LIN {X 0,Y 425.438,Z 376.705,A -85,B 0,C 180,E1 18577.302,E2 18577.302} C_VEL
LIN {X 0,Y 425.151,Z 380.959,A -85,B 0,C 180,E1 18577.085,E2 18577.085} C_VEL
LIN {X 0,Y 415.891,Z 452.689,A -85,B 0,C 180,E1 18574.855,E2 18574.855} C_VEL
LIN {X 0,Y 409.352,Z 519.498,A -85,B 0,C 180,E1 18572.849,E2 18572.849} C_VEL
LIN {X 0,Y 405.386,Z 570.426,A -85,B 0,C 180,E1 18571.36,E2 18571.36} C_VEL
LIN {X 0,Y 403.425,Z 591.228,A -85,B 0,C 180,E1 18570.479,E2 18570.479} C_VEL
LIN {X 0,Y 401.306,Z 610.6,A -85,B 0,C 180,E1 18569.395,E2 18569.395} C_VEL
LIN {X 0,Y 398.96,Z 629.842,A -85,B 0,C 180,E1 18568.028,E2 18568.028} C_VEL
LIN {X 0,Y 396.521,Z 647.903,A -85,B 0,C 180,E1 18566.427,E2 18566.427} C_VEL
LIN {X 0,Y 394.184,Z 664.215,A -85,B 0,C 180,E1 18564.661,E2 18564.661} C_VEL
LIN {X 0,Y 391.906,Z 679.493,A -85,B 0,C 180,E1 18562.658,E2 18562.658} C_VEL
LIN {X 0,Y 389.92,Z 692.735,A -85,B 0,C 180,E1 18560.567,E2 18560.567} C_VEL
LIN {X 0,Y 388.182,Z 704.572,A -85,B 0,C 180,E1 18558.315,E2 18558.315} C_VEL
LIN {X 0,Y 386.73,Z 715.054,A -85,B 0,C 180,E1 18555.89,E2 18555.89} C_VEL
LIN {X 0,Y 385.62,Z 723.955,A -85,B 0,C 180,E1 18553.342,E2 18553.342} C_VEL
LIN {X 0,Y 384.866,Z 731.025,A -85,B 0,C 180,E1 18550.78,E2 18550.78} C_VEL
LIN {X 0,Y 384.39,Z 736.661,A -85,B 0,C 180,E1 18548.074,E2 18548.074} C_VEL
LIN {X 0,Y 384.156,Z 740.555,A -85,B 0,C 180,E1 18545.376,E2 18545.376} C_VEL
LIN {X 0,Y 384.055,Z 742.806,A -85,B 0,C 180,E1 18542.685,E2 18542.685} C_VEL
LIN {X 0,Y 384.034,Z 743.462,A -85,B 0,C 180,E1 18539.999,E2 18539.999} C_VEL
LIN {X 0,Y 384.039,Z 742.418,A -85,B 0,C 180,E1 18537.164,E2 18537.164} C_VEL
LIN {X 0,Y 384.119,Z 739.593,A -85,B 0,C 180,E1 18534.323,E2 18534.323} C_VEL
LIN {X 0,Y 384.335,Z 735.21,A -85,B 0,C 180,E1 18531.622,E2 18531.622} C_VEL
LIN {X 0,Y 384.782,Z 729.053,A -85,B 0,C 180,E1 18528.913,E2 18528.913} C_VEL
LIN {X 0,Y 385.56,Z 720.955,A -85,B 0,C 180,E1 18526.197,E2 18526.197} C_VEL
LIN {X 0,Y 386.687,Z 711.151,A -85,B 0,C 180,E1 18523.599,E2 18523.599} C_VEL
LIN {X 0,Y 388.11,Z 700.088,A -85,B 0,C 180,E1 18521.214,E2 18521.214} C_VEL
LIN {X 0,Y 389.844,Z 687.4,A -85,B 0,C 180,E1 18518.956,E2 18518.956} C_VEL
LIN {X 0,Y 391.826,Z 673.161,A -85,B 0,C 180,E1 18516.86,E2 18516.86} C_VEL
LIN {X 0,Y 393.943,Z 657.683,A -85,B 0,C 180,E1 18514.973,E2 18514.973} C_VEL
LIN {X 0,Y 396.1,Z 640.996,A -85,B 0,C 180,E1 18513.299,E2 18513.299} C_VEL
LIN {X 0,Y 398.237,Z 622.993,A -85,B 0,C 180,E1 18511.834,E2 18511.834} C_VEL
LIN {X 0,Y 400.237,Z 603.839,A -85,B 0,C 180,E1 18510.6,E2 18510.6} C_VEL
LIN {X 0,Y 401.921,Z 584.234,A -85,B 0,C 180,E1 18509.637,E2 18509.637} C_VEL
LIN {X 0,Y 403.261,Z 564.613,A -85,B 0,C 180,E1 18508.948,E2 18508.948} C_VEL
LIN {X 0,Y 404.762,Z 527.661,A -85,B 0,C 180,E1 18508.112,E2 18508.112} C_VEL
LIN {X 0,Y 410.951,Z 374.818,A -85,B 0,C 180,E1 18504.8,E2 18504.8} C_VEL
LIN {X 0,Y 406.023,Z 341.792,A -85,B 0,C 180,E1 18503.459,E2 18503.459} C_VEL
LIN {X 0,Y 404.74,Z 338.868,A -85,B 0,C 180,E1 18503.17,E2 18503.17} C_VEL
LIN {X 0,Y 398.098,Z 320.346,A -85,B 0,C 180,E1 18500.225,E2 18500.225} C_VEL
LIN {X 0,Y 390.871,Z 301.781,A -85,B 0,C 180,E1 18497.022,E2 18497.022} C_VEL
LIN {X 0,Y 385.651,Z 288.651,A -85,B 0,C 180,E1 18494.544,E2 18494.544} C_VEL
LIN {X 0,Y 385.626,Z 288.452,A -85,B 0,C 180,E1 18490.562,E2 18490.562} C_VEL
LIN {X 0,Y 385.621,Z 288.448,A -85,B 0,C 180,E1 18486.506,E2 18486.506} C_VEL
LIN {X 0,Y 385.621,Z 288.449,A -85,B 0,C 180,E1 18482.462,E2 18482.462} C_VEL
LIN {X 0,Y 385.618,Z 288.434,A -85,B 0,C 180,E1 18478.479,E2 18478.479} C_VEL
LIN {X 0,Y 385.609,Z 288.434,A -85,B 0,C 180,E1 18474.476,E2 18474.476} C_VEL
LIN {X 0,Y 385.596,Z 288.441,A -85,B 0,C 180,E1 18470.595,E2 18470.595} C_VEL
LIN {X 0,Y 385.63,Z 288.664,A -85,B 0,C 180,E1 18469.542,E2 18469.542} C_VEL
LIN {X 0,Y 388.127,Z 294.947,A -85,B 0,C 180,E1 18468.554,E2 18468.554} C_VEL
LIN {X 0,Y 395.619,Z 313.822,A -85,B 0,C 180,E1 18465.841,E2 18465.841} C_VEL
LIN {X 0,Y 402.27,Z 333.616,A -85,B 0,C 180,E1 18463.22,E2 18463.22} C_VEL
LIN {X 0,Y 402.753,Z 336.308,A -85,B 0,C 180,E1 18462.912,E2 18462.912} C_VEL
LIN {X 0,Y 402.207,Z 346.122,A -85,B 0,C 180,E1 18462.001,E2 18462.001} C_VEL
LIN {X 0,Y 400.979,Z 352.785,A -85,B 0,C 180,E1 18461.461,E2 18461.461} C_VEL
LIN {X 0,Y 394.437,Z 371.147,A -85,B 0,C 180,E1 18460.234,E2 18460.234} C_VEL
LIN {X 0,Y 393.42,Z 376.867,A -85,B 0,C 180,E1 18459.755,E2 18459.755} C_VEL
LIN {X 0,Y 390.87,Z 418.201,A -85,B 0,C 180,E1 18455.874,E2 18455.874} C_VEL
LIN {X 0,Y 388.343,Z 461.181,A -85,B 0,C 180,E1 18451.846,E2 18451.846} C_VEL
LIN {X 0,Y 387.324,Z 479.827,A -85,B 0,C 180,E1 18450.126,E2 18450.126} C_VEL
LIN {X 0,Y 389.149,Z 497.663,A -85,B 0,C 180,E1 18449.64,E2 18449.64} C_VEL
LIN {X 0,Y 386.608,Z 623.155,A -85,B 0,C 180,E1 18447.245,E2 18447.245} C_VEL
LIN {X 0,Y 385.965,Z 639.192,A -85,B 0,C 180,E1 18446.667,E2 18446.667} C_VEL
LIN {X 0,Y 384.984,Z 655.233,A -85,B 0,C 180,E1 18445.801,E2 18445.801} C_VEL
LIN {X 0,Y 383.849,Z 669.257,A -85,B 0,C 180,E1 18444.771,E2 18444.771} C_VEL
LIN {X 0,Y 382.459,Z 683.671,A -85,B 0,C 180,E1 18443.396,E2 18443.396} C_VEL
LIN {X 0,Y 381.091,Z 696.381,A -85,B 0,C 180,E1 18441.857,E2 18441.857} C_VEL
LIN {X 0,Y 379.695,Z 708.569,A -85,B 0,C 180,E1 18439.993,E2 18439.993} C_VEL
LIN {X 0,Y 378.562,Z 718.372,A -85,B 0,C 180,E1 18438.113,E2 18438.113} C_VEL
LIN {X 0,Y 377.555,Z 727.448,A -85,B 0,C 180,E1 18435.901,E2 18435.901} C_VEL
LIN {X 0,Y 376.862,Z 734.493,A -85,B 0,C 180,E1 18433.668,E2 18433.668} C_VEL
LIN {X 0,Y 376.406,Z 740.037,A -85,B 0,C 180,E1 18431.253,E2 18431.253} C_VEL
LIN {X 0,Y 376.179,Z 743.765,A -85,B 0,C 180,E1 18428.811,E2 18428.811} C_VEL
LIN {X 0,Y 376.095,Z 745.698,A -85,B 0,C 180,E1 18426.334,E2 18426.334} C_VEL
LIN {X 0,Y 376.098,Z 745.901,A -85,B 0,C 180,E1 18423.815,E2 18423.815} C_VEL
LIN {X 0,Y 376.188,Z 744.18,A -85,B 0,C 180,E1 18421.247,E2 18421.247} C_VEL
LIN {X 0,Y 376.427,Z 740.771,A -85,B 0,C 180,E1 18418.793,E2 18418.793} C_VEL
LIN {X 0,Y 376.894,Z 735.364,A -85,B 0,C 180,E1 18416.329,E2 18416.329} C_VEL
LIN {X 0,Y 377.598,Z 728.744,A -85,B 0,C 180,E1 18414.124,E2 18414.124} C_VEL
LIN {X 0,Y 378.619,Z 719.95,A -85,B 0,C 180,E1 18411.904,E2 18411.904} C_VEL
LIN {X 0,Y 379.783,Z 710.471,A -85,B 0,C 180,E1 18410.008,E2 18410.008} C_VEL
LIN {X 0,Y 381.141,Z 699.241,A -85,B 0,C 180,E1 18408.219,E2 18408.219} C_VEL
LIN {X 0,Y 382.607,Z 686.432,A -85,B 0,C 180,E1 18406.587,E2 18406.587} C_VEL
LIN {X 0,Y 383.966,Z 673.167,A -85,B 0,C 180,E1 18405.254,E2 18405.254} C_VEL
LIN {X 0,Y 385.314,Z 657.803,A -85,B 0,C 180,E1 18404.063,E2 18404.063} C_VEL
LIN {X 0,Y 386.332,Z 642.25,A -85,B 0,C 180,E1 18403.18,E2 18403.18} C_VEL
LIN {X 0,Y 387.065,Z 625.559,A -85,B 0,C 180,E1 18402.536,E2 18402.536} C_VEL
LIN {X 0,Y 387.736,Z 593.398,A -85,B 0,C 180,E1 18401.872,E2 18401.872} C_VEL
LIN {X 0,Y 389.648,Z 494.75,A -85,B 0,C 180,E1 18399.99,E2 18399.99} C_VEL
LIN {X 0,Y 387.952,Z 480.003,A -85,B 0,C 180,E1 18399.539,E2 18399.539} C_VEL
LIN {X 0,Y 390.482,Z 436.326,A -85,B 0,C 180,E1 18395.489,E2 18395.489} C_VEL
LIN {X 0,Y 393.042,Z 393.106,A -85,B 0,C 180,E1 18391.487,E2 18391.487} C_VEL
LIN {X 0,Y 395.389,Z 349.348,A -85,B 0,C 180,E1 18387.485,E2 18387.485} C_VEL
LIN {X 0,Y 396.024,Z 337.35,A -85,B 0,C 180,E1 18386.383,E2 18386.383} C_VEL
LIN {X 0,Y 390.695,Z 320.827,A -85,B 0,C 180,E1 18384.172,E2 18384.172} C_VEL
LIN {X 0,Y 384.015,Z 303.953,A -85,B 0,C 180,E1 18381.699,E2 18381.699} C_VEL
LIN {X 0,Y 378.89,Z 292.803,A -85,B 0,C 180,E1 18379.903,E2 18379.903} C_VEL
LIN {X 0,Y 377.731,Z 289.764,A -85,B 0,C 180,E1 18379.363,E2 18379.363} C_VEL
LIN {X 0,Y 377.654,Z 289.433,A -85,B 0,C 180,E1 18378.205,E2 18378.205} C_VEL
LIN {X 0,Y 377.653,Z 289.441,A -85,B 0,C 180,E1 18374.255,E2 18374.255} C_VEL
LIN {X 0,Y 377.653,Z 289.443,A -85,B 0,C 180,E1 18370.218,E2 18370.218} C_VEL
LIN {X 0,Y 377.652,Z 289.439,A -85,B 0,C 180,E1 18366.232,E2 18366.232} C_VEL
LIN {X 0,Y 377.652,Z 289.442,A -85,B 0,C 180,E1 18362.125,E2 18362.125} C_VEL
LIN {X 0,Y 377.653,Z 289.439,A -85,B 0,C 180,E1 18358.18,E2 18358.18} C_VEL
LIN {X 0,Y 377.655,Z 289.443,A -85,B 0,C 180,E1 18354.074,E2 18354.074} C_VEL
LIN {X 0,Y 377.655,Z 289.435,A -85,B 0,C 180,E1 18350.012,E2 18350.012} C_VEL
LIN {X 0,Y 377.658,Z 289.442,A -85,B 0,C 180,E1 18345.903,E2 18345.903} C_VEL
LIN {X 0,Y 377.661,Z 289.44,A -85,B 0,C 180,E1 18341.796,E2 18341.796} C_VEL
LIN {X 0,Y 377.66,Z 289.436,A -85,B 0,C 180,E1 18337.754,E2 18337.754} C_VEL
LIN {X 0,Y 377.662,Z 289.443,A -85,B 0,C 180,E1 18333.76,E2 18333.76} C_VEL
LIN {X 0,Y 377.663,Z 289.438,A -85,B 0,C 180,E1 18329.8,E2 18329.8} C_VEL
LIN {X 0,Y 377.664,Z 289.439,A -85,B 0,C 180,E1 18325.674,E2 18325.674} C_VEL
LIN {X 0,Y 377.666,Z 289.44,A -85,B 0,C 180,E1 18321.592,E2 18321.592} C_VEL
LIN {X 0,Y 377.716,Z 289.737,A -85,B 0,C 180,E1 18319.409,E2 18319.409} C_VEL
LIN {X 0,Y 386.088,Z 309.298,A -85,B 0,C 180,E1 18315.843,E2 18315.843} C_VEL
LIN {X 0,Y 390.517,Z 319.683,A -85,B 0,C 180,E1 18314.145,E2 18314.145} C_VEL
LIN {X 0,Y 407.06,Z 348.807,A -85,B 0,C 180,E1 18311.54,E2 18311.54} C_VEL
LIN {X 0,Y 409.737,Z 354.251,A -85,B 0,C 180,E1 18311.13,E2 18311.13} C_VEL
LIN {X 0,Y 401.571,Z 543.738,A -85,B 0,C 180,E1 18307.075,E2 18307.075} C_VEL
LIN {X 0,Y 399.995,Z 579.391,A -85,B 0,C 180,E1 18306.266,E2 18306.266} C_VEL
LIN {X 0,Y 398.438,Z 600.282,A -85,B 0,C 180,E1 18305.547,E2 18305.547} C_VEL
LIN {X 0,Y 396.573,Z 619.61,A -85,B 0,C 180,E1 18304.646,E2 18304.646} C_VEL
LIN {X 0,Y 394.235,Z 640.263,A -85,B 0,C 180,E1 18303.389,E2 18303.389} C_VEL
LIN {X 0,Y 391.688,Z 659.766,A -85,B 0,C 180,E1 18301.895,E2 18301.895} C_VEL
LIN {X 0,Y 389.061,Z 678.211,A -85,B 0,C 180,E1 18300.158,E2 18300.158} C_VEL
LIN {X 0,Y 386.426,Z 695.615,A -85,B 0,C 180,E1 18298.176,E2 18298.176} C_VEL
LIN {X 0,Y 384.038,Z 711.023,A -85,B 0,C 180,E1 18296.075,E2 18296.075} C_VEL
LIN {X 0,Y 381.869,Z 725.235,A -85,B 0,C 180,E1 18293.778,E2 18293.778} C_VEL
LIN {X 0,Y 379.977,Z 738.176,A -85,B 0,C 180,E1 18291.29,E2 18291.29} C_VEL
LIN {X 0,Y 378.451,Z 749.682,A -85,B 0,C 180,E1 18288.641,E2 18288.641} C_VEL
LIN {X 0,Y 377.326,Z 759.627,A -85,B 0,C 180,E1 18285.869,E2 18285.869} C_VEL
LIN {X 0,Y 376.568,Z 767.994,A -85,B 0,C 180,E1 18282.98,E2 18282.98} C_VEL
LIN {X 0,Y 376.163,Z 774.767,A -85,B 0,C 180,E1 18279.947,E2 18279.947} C_VEL
LIN {X 0,Y 376.018,Z 779.281,A -85,B 0,C 180,E1 18277.178,E2 18277.178} C_VEL
LIN {X 0,Y 376.01,Z 782.442,A -85,B 0,C 180,E1 18274.268,E2 18274.268} C_VEL
LIN {X 0,Y 376.025,Z 784,A -85,B 0,C 180,E1 18271.37,E2 18271.37} C_VEL
LIN {X 0,Y 376.03,Z 783.923,A -85,B 0,C 180,E1 18268.627,E2 18268.627} C_VEL
LIN {X 0,Y 376.014,Z 782.237,A -85,B 0,C 180,E1 18265.679,E2 18265.679} C_VEL
LIN {X 0,Y 376.027,Z 778.801,A -85,B 0,C 180,E1 18262.666,E2 18262.666} C_VEL
LIN {X 0,Y 376.183,Z 774.096,A -85,B 0,C 180,E1 18259.895,E2 18259.895} C_VEL
LIN {X 0,Y 376.573,Z 767.289,A -85,B 0,C 180,E1 18256.955,E2 18256.955} C_VEL
LIN {X 0,Y 377.294,Z 759.002,A -85,B 0,C 180,E1 18254.148,E2 18254.148} C_VEL
LIN {X 0,Y 378.404,Z 748.838,A -85,B 0,C 180,E1 18251.353,E2 18251.353} C_VEL
LIN {X 0,Y 380.005,Z 736.395,A -85,B 0,C 180,E1 18248.546,E2 18248.546} C_VEL
LIN {X 0,Y 381.94,Z 722.847,A -85,B 0,C 180,E1 18246.011,E2 18246.011} C_VEL
LIN {X 0,Y 384.155,Z 708.03,A -85,B 0,C 180,E1 18243.683,E2 18243.683} C_VEL
LIN {X 0,Y 386.6,Z 691.972,A -85,B 0,C 180,E1 18241.562,E2 18241.562} C_VEL
LIN {X 0,Y 389.239,Z 674.193,A -85,B 0,C 180,E1 18239.598,E2 18239.598} C_VEL
LIN {X 0,Y 391.918,Z 655.491,A -85,B 0,C 180,E1 18237.886,E2 18237.886} C_VEL
LIN {X 0,Y 394.591,Z 635.281,A -85,B 0,C 180,E1 18236.373,E2 18236.373} C_VEL
LIN {X 0,Y 397.071,Z 614.668,A -85,B 0,C 180,E1 18235.136,E2 18235.136} C_VEL
LIN {X 0,Y 399.349,Z 593.081,A -85,B 0,C 180,E1 18234.134,E2 18234.134} C_VEL
LIN {X 0,Y 401.355,Z 570.136,A -85,B 0,C 180,E1 18233.363,E2 18233.363} C_VEL
LIN {X 0,Y 406.419,Z 500.604,A -85,B 0,C 180,E1 18231.493,E2 18231.493} C_VEL
LIN {X 0,Y 412.494,Z 440.99,A -85,B 0,C 180,E1 18229.737,E2 18229.737} C_VEL
LIN {X 0,Y 420.617,Z 380.86,A -85,B 0,C 180,E1 18227.859,E2 18227.859} C_VEL
LIN {X 0,Y 423.847,Z 360.47,A -85,B 0,C 180,E1 18227.193,E2 18227.193} C_VEL
LIN {X 0,Y 422.14,Z 356.085,A -85,B 0,C 180,E1 18225.959,E2 18225.959} C_VEL
LIN {X 0,Y 420.779,Z 353.237,A -85,B 0,C 180,E1 18224.315,E2 18224.315} C_VEL
LIN {X 0,Y 420.316,Z 353.415,A -85,B 0,C 180,E1 18223.286,E2 18223.286} C_VEL
LIN {X 0,Y 420.495,Z 355.616,A -85,B 0,C 180,E1 18221.699,E2 18221.699} C_VEL
LIN {X 0,Y 421.439,Z 359.627,A -85,B 0,C 180,E1 18220.301,E2 18220.301} C_VEL
LIN {X 0,Y 422.49,Z 363.795,A -85,B 0,C 180,E1 18219.315,E2 18219.315} C_VEL
LIN {X 0,Y 421.522,Z 380.833,A -85,B 0,C 180,E1 18218.088,E2 18218.088} C_VEL
LIN {X 0,Y 411.493,Z 450.143,A -85,B 0,C 180,E1 18215.839,E2 18215.839} C_VEL
LIN {X 0,Y 404.087,Z 516.008,A -85,B 0,C 180,E1 18213.767,E2 18213.767} C_VEL
LIN {X 0,Y 399.163,Z 571.366,A -85,B 0,C 180,E1 18212.064,E2 18212.064} C_VEL
LIN {X 0,Y 397.052,Z 591.572,A -85,B 0,C 180,E1 18211.176,E2 18211.176} C_VEL
LIN {X 0,Y 394.706,Z 611.287,A -85,B 0,C 180,E1 18210.041,E2 18210.041} C_VEL
LIN {X 0,Y 392.165,Z 630.471,A -85,B 0,C 180,E1 18208.641,E2 18208.641} C_VEL
LIN {X 0,Y 389.562,Z 648.351,A -85,B 0,C 180,E1 18207.019,E2 18207.019} C_VEL
LIN {X 0,Y 387.063,Z 664.574,A -85,B 0,C 180,E1 18205.228,E2 18205.228} C_VEL
LIN {X 0,Y 384.714,Z 679.307,A -85,B 0,C 180,E1 18203.268,E2 18203.268} C_VEL
LIN {X 0,Y 382.565,Z 692.626,A -85,B 0,C 180,E1 18201.141,E2 18201.141} C_VEL
LIN {X 0,Y 380.677,Z 704.546,A -85,B 0,C 180,E1 18198.848,E2 18198.848} C_VEL
LIN {X 0,Y 379.096,Z 715.051,A -85,B 0,C 180,E1 18196.392,E2 18196.392} C_VEL
LIN {X 0,Y 377.852,Z 724.092,A -85,B 0,C 180,E1 18193.777,E2 18193.777} C_VEL
LIN {X 0,Y 376.99,Z 731.413,A -85,B 0,C 180,E1 18191.088,E2 18191.088} C_VEL
LIN {X 0,Y 376.472,Z 736.951,A -85,B 0,C 180,E1 18188.399,E2 18188.399} C_VEL
LIN {X 0,Y 376.195,Z 740.911,A -85,B 0,C 180,E1 18185.643,E2 18185.643} C_VEL
LIN {X 0,Y 376.078,Z 743.22,A -85,B 0,C 180,E1 18182.895,E2 18182.895} C_VEL
LIN {X 0,Y 376.045,Z 743.906,A -85,B 0,C 180,E1 18180.152,E2 18180.152} C_VEL
LIN {X 0,Y 376.045,Z 742.986,A -85,B 0,C 180,E1 18177.409,E2 18177.409} C_VEL
LIN {X 0,Y 376.115,Z 740.47,A -85,B 0,C 180,E1 18174.661,E2 18174.661} C_VEL
LIN {X 0,Y 376.317,Z 736.296,A -85,B 0,C 180,E1 18171.904,E2 18171.904} C_VEL
LIN {X 0,Y 376.755,Z 730.362,A -85,B 0,C 180,E1 18169.139,E2 18169.139} C_VEL
LIN {X 0,Y 377.502,Z 722.694,A -85,B 0,C 180,E1 18166.424,E2 18166.424} C_VEL
LIN {X 0,Y 378.557,Z 713.707,A -85,B 0,C 180,E1 18163.898,E2 18163.898} C_VEL
LIN {X 0,Y 379.979,Z 702.936,A -85,B 0,C 180,E1 18161.434,E2 18161.434} C_VEL
LIN {X 0,Y 381.705,Z 690.726,A -85,B 0,C 180,E1 18159.13,E2 18159.13} C_VEL
LIN {X 0,Y 383.685,Z 677.062,A -85,B 0,C 180,E1 18156.989,E2 18156.989} C_VEL
LIN {X 0,Y 385.869,Z 661.873,A -85,B 0,C 180,E1 18155.015,E2 18155.015} C_VEL
LIN {X 0,Y 388.085,Z 645.73,A -85,B 0,C 180,E1 18153.283,E2 18153.283} C_VEL
LIN {X 0,Y 390.283,Z 628.511,A -85,B 0,C 180,E1 18151.769,E2 18151.769} C_VEL
LIN {X 0,Y 392.391,Z 609.893,A -85,B 0,C 180,E1 18150.455,E2 18150.455} C_VEL
LIN {X 0,Y 394.273,Z 590.391,A -85,B 0,C 180,E1 18149.391,E2 18149.391} C_VEL
LIN {X 0,Y 395.803,Z 570.164,A -85,B 0,C 180,E1 18148.588,E2 18148.588} C_VEL
LIN {X 0,Y 396.936,Z 548.319,A -85,B 0,C 180,E1 18148.015,E2 18148.015} C_VEL
LIN {X 0,Y 404.242,Z 376.052,A -85,B 0,C 180,E1 18144.2,E2 18144.2} C_VEL
LIN {X 0,Y 399.757,Z 345.342,A -85,B 0,C 180,E1 18142.929,E2 18142.929} C_VEL
LIN {X 0,Y 396.829,Z 339.435,A -85,B 0,C 180,E1 18142.428,E2 18142.428} C_VEL
LIN {X 0,Y 389.659,Z 319.65,A -85,B 0,C 180,E1 18139.199,E2 18139.199} C_VEL
LIN {X 0,Y 382.005,Z 300.218,A -85,B 0,C 180,E1 18135.715,E2 18135.715} C_VEL
LIN {X 0,Y 377.705,Z 289.65,A -85,B 0,C 180,E1 18133.635,E2 18133.635} C_VEL
LIN {X 0,Y 377.684,Z 289.439,A -85,B 0,C 180,E1 18129.611,E2 18129.611} C_VEL
LIN {X 0,Y 377.682,Z 289.441,A -85,B 0,C 180,E1 18125.622,E2 18125.622} C_VEL
LIN {X 0,Y 377.683,Z 289.439,A -85,B 0,C 180,E1 18121.52,E2 18121.52} C_VEL
LIN {X 0,Y 377.673,Z 289.44,A -85,B 0,C 180,E1 18117.431,E2 18117.431} C_VEL
LIN {X 0,Y 377.665,Z 289.439,A -85,B 0,C 180,E1 18113.4,E2 18113.4} C_VEL
LIN {X 0,Y 377.702,Z 289.655,A -85,B 0,C 180,E1 18110.353,E2 18110.353} C_VEL
LIN {X 0,Y 385.933,Z 309.834,A -85,B 0,C 180,E1 18107.257,E2 18107.257} C_VEL
LIN {X 0,Y 392.695,Z 328.668,A -85,B 0,C 180,E1 18104.637,E2 18104.637} C_VEL
LIN {X 0,Y 395.707,Z 338.188,A -85,B 0,C 180,E1 18103.39,E2 18103.39} C_VEL
LIN {X 0,Y 393.42,Z 376.867,A -85,B 0,C 180,E1 18099.755,E2 18099.755} C_VEL
LIN {X 0,Y 392.128,Z 383.541,A -85,B 0,C 180,E1 18099.208,E2 18099.208} C_VEL
LIN {X 0,Y 385.455,Z 401.884,A -85,B 0,C 180,E1 18097.961,E2 18097.961} C_VEL
LIN {X 0,Y 384.433,Z 407.611,A -85,B 0,C 180,E1 18097.475,E2 18097.475} C_VEL
LIN {X 0,Y 381.606,Z 451.549,A -85,B 0,C 180,E1 18093.306,E2 18093.306} C_VEL
LIN {X 0,Y 379.974,Z 480.131,A -85,B 0,C 180,E1 18090.629,E2 18090.629} C_VEL
LIN {X 0,Y 381.841,Z 498.458,A -85,B 0,C 180,E1 18090.116,E2 18090.116} C_VEL
LIN {X 0,Y 379.17,Z 623.534,A -85,B 0,C 180,E1 18087.683,E2 18087.683} C_VEL
LIN {X 0,Y 378.494,Z 639.636,A -85,B 0,C 180,E1 18087.091,E2 18087.091} C_VEL
LIN {X 0,Y 377.466,Z 655.734,A -85,B 0,C 180,E1 18086.205,E2 18086.205} C_VEL
LIN {X 0,Y 376.243,Z 670.094,A -85,B 0,C 180,E1 18085.123,E2 18085.123} C_VEL
LIN {X 0,Y 374.792,Z 684.434,A -85,B 0,C 180,E1 18083.722,E2 18083.722} C_VEL
LIN {X 0,Y 373.359,Z 697.059,A -85,B 0,C 180,E1 18082.152,E2 18082.152} C_VEL
LIN {X 0,Y 371.897,Z 709.206,A -85,B 0,C 180,E1 18080.25,E2 18080.25} C_VEL
LIN {X 0,Y 370.678,Z 719.166,A -85,B 0,C 180,E1 18078.282,E2 18078.282} C_VEL
LIN {X 0,Y 369.647,Z 727.998,A -85,B 0,C 180,E1 18076.072,E2 18076.072} C_VEL
LIN {X 0,Y 368.914,Z 734.996,A -85,B 0,C 180,E1 18073.792,E2 18073.792} C_VEL
LIN {X 0,Y 368.428,Z 740.585,A -85,B 0,C 180,E1 18071.289,E2 18071.289} C_VEL
LIN {X 0,Y 368.192,Z 744.202,A -85,B 0,C 180,E1 18068.83,E2 18068.83} C_VEL
LIN {X 0,Y 368.104,Z 746.127,A -85,B 0,C 180,E1 18066.261,E2 18066.261} C_VEL
LIN {X 0,Y 368.109,Z 746.272,A -85,B 0,C 180,E1 18063.723,E2 18063.723} C_VEL
LIN {X 0,Y 368.211,Z 744.521,A -85,B 0,C 180,E1 18061.098,E2 18061.098} C_VEL
LIN {X 0,Y 368.472,Z 741.087,A -85,B 0,C 180,E1 18058.603,E2 18058.603} C_VEL
LIN {X 0,Y 368.99,Z 735.613,A -85,B 0,C 180,E1 18056.071,E2 18056.071} C_VEL
LIN {X 0,Y 369.729,Z 729.147,A -85,B 0,C 180,E1 18053.879,E2 18053.879} C_VEL
LIN {X 0,Y 370.786,Z 720.614,A -85,B 0,C 180,E1 18051.671,E2 18051.671} C_VEL
LIN {X 0,Y 372.085,Z 710.69,A -85,B 0,C 180,E1 18049.641,E2 18049.641} C_VEL
LIN {X 0,Y 373.545,Z 699.243,A -85,B 0,C 180,E1 18047.793,E2 18047.793} C_VEL
LIN {X 0,Y 375.103,Z 686.352,A -85,B 0,C 180,E1 18046.131,E2 18046.131} C_VEL
LIN {X 0,Y 376.6,Z 672.251,A -85,B 0,C 180,E1 18044.715,E2 18044.715} C_VEL
LIN {X 0,Y 377.97,Z 657.195,A -85,B 0,C 180,E1 18043.549,E2 18043.549} C_VEL
LIN {X 0,Y 379.05,Z 640.978,A -85,B 0,C 180,E1 18042.641,E2 18042.641} C_VEL
LIN {X 0,Y 379.755,Z 624.876,A -85,B 0,C 180,E1 18042.033,E2 18042.033} C_VEL
LIN {X 0,Y 381.195,Z 558.96,A -85,B 0,C 180,E1 18040.716,E2 18040.716} C_VEL
LIN {X 0,Y 382.467,Z 495.618,A -85,B 0,C 180,E1 18039.476,E2 18039.476} C_VEL
LIN {X 0,Y 380.711,Z 480.143,A -85,B 0,C 180,E1 18038.982,E2 18038.982} C_VEL
LIN {X 0,Y 383.378,Z 436.859,A -85,B 0,C 180,E1 18034.923,E2 18034.923} C_VEL
LIN {X 0,Y 385.959,Z 395.249,A -85,B 0,C 180,E1 18031.033,E2 18031.033} C_VEL
LIN {X 0,Y 388.328,Z 354.742,A -85,B 0,C 180,E1 18027.279,E2 18027.279} C_VEL
LIN {X 0,Y 389.068,Z 340.012,A -85,B 0,C 180,E1 18025.906,E2 18025.906} C_VEL
LIN {X 0,Y 383.738,Z 323.637,A -85,B 0,C 180,E1 18023.658,E2 18023.658} C_VEL
LIN {X 0,Y 377.887,Z 308.744,A -85,B 0,C 180,E1 18021.417,E2 18021.417} C_VEL
LIN {X 0,Y 371.317,Z 294.299,A -85,B 0,C 180,E1 18019.016,E2 18019.016} C_VEL
LIN {X 0,Y 369.768,Z 290.793,A -85,B 0,C 180,E1 18018.365,E2 18018.365} C_VEL
LIN {X 0,Y 369.741,Z 290.423,A -85,B 0,C 180,E1 18017.631,E2 18017.631} C_VEL
LIN {X 0,Y 369.751,Z 290.433,A -85,B 0,C 180,E1 18013.448,E2 18013.448} C_VEL
LIN {X 0,Y 369.746,Z 290.428,A -85,B 0,C 180,E1 18009.255,E2 18009.255} C_VEL
LIN {X 0,Y 369.746,Z 290.43,A -85,B 0,C 180,E1 18005.276,E2 18005.276} C_VEL
LIN {X 0,Y 369.746,Z 290.425,A -85,B 0,C 180,E1 18001.085,E2 18001.085} C_VEL
LIN {X 0,Y 369.741,Z 290.427,A -85,B 0,C 180,E1 17997.055,E2 17997.055} C_VEL
LIN {X 0,Y 369.746,Z 290.423,A -85,B 0,C 180,E1 17992.927,E2 17992.927} C_VEL
LIN {X 0,Y 369.735,Z 290.429,A -85,B 0,C 180,E1 17988.773,E2 17988.773} C_VEL
LIN {X 0,Y 369.742,Z 290.423,A -85,B 0,C 180,E1 17984.793,E2 17984.793} C_VEL
LIN {X 0,Y 369.737,Z 290.424,A -85,B 0,C 180,E1 17980.689,E2 17980.689} C_VEL
LIN {X 0,Y 369.735,Z 290.429,A -85,B 0,C 180,E1 17976.577,E2 17976.577} C_VEL
LIN {X 0,Y 369.731,Z 290.426,A -85,B 0,C 180,E1 17972.456,E2 17972.456} C_VEL
LIN {X 0,Y 369.733,Z 290.427,A -85,B 0,C 180,E1 17968.408,E2 17968.408} C_VEL
LIN {X 0,Y 369.727,Z 290.428,A -85,B 0,C 180,E1 17964.259,E2 17964.259} C_VEL
LIN {X 0,Y 369.775,Z 290.691,A -85,B 0,C 180,E1 17960.413,E2 17960.413} C_VEL
LIN {X 0,Y 372.529,Z 297.351,A -85,B 0,C 180,E1 17959.089,E2 17959.089} C_VEL
LIN {X 0,Y 380.514,Z 315.687,A -85,B 0,C 180,E1 17955.762,E2 17955.762} C_VEL
LIN {X 0,Y 382.502,Z 320.216,A -85,B 0,C 180,E1 17955.055,E2 17955.055} C_VEL
LIN {X 0,Y 398.543,Z 348.214,A -85,B 0,C 180,E1 17952.448,E2 17952.448} C_VEL
LIN {X 0,Y 403.094,Z 356.879,A -85,B 0,C 180,E1 17951.729,E2 17951.729} C_VEL
LIN {X 0,Y 394.051,Z 557.218,A -85,B 0,C 180,E1 17947.35,E2 17947.35} C_VEL
LIN {X 0,Y 392.751,Z 582.341,A -85,B 0,C 180,E1 17946.724,E2 17946.724} C_VEL
LIN {X 0,Y 390.974,Z 603.771,A -85,B 0,C 180,E1 17945.93,E2 17945.93} C_VEL
LIN {X 0,Y 388.828,Z 624.372,A -85,B 0,C 180,E1 17944.886,E2 17944.886} C_VEL
LIN {X 0,Y 386.349,Z 644.626,A -85,B 0,C 180,E1 17943.559,E2 17943.559} C_VEL
LIN {X 0,Y 383.787,Z 663.16,A -85,B 0,C 180,E1 17942.05,E2 17942.05} C_VEL
LIN {X 0,Y 381.235,Z 680.303,A -85,B 0,C 180,E1 17940.361,E2 17940.361} C_VEL
LIN {X 0,Y 378.598,Z 697.08,A -85,B 0,C 180,E1 17938.381,E2 17938.381} C_VEL
LIN {X 0,Y 376.01,Z 713.155,A -85,B 0,C 180,E1 17936.107,E2 17936.107} C_VEL
LIN {X 0,Y 373.725,Z 727.589,A -85,B 0,C 180,E1 17933.658,E2 17933.658} C_VEL
LIN {X 0,Y 371.736,Z 740.831,A -85,B 0,C 180,E1 17930.959,E2 17930.959} C_VEL
LIN {X 0,Y 370.249,Z 751.822,A -85,B 0,C 180,E1 17928.254,E2 17928.254} C_VEL
LIN {X 0,Y 369.161,Z 761.382,A -85,B 0,C 180,E1 17925.39,E2 17925.39} C_VEL
LIN {X 0,Y 368.458,Z 769.429,A -85,B 0,C 180,E1 17922.377,E2 17922.377} C_VEL
LIN {X 0,Y 368.119,Z 775.579,A -85,B 0,C 180,E1 17919.377,E2 17919.377} C_VEL
LIN {X 0,Y 368.022,Z 779.808,A -85,B 0,C 180,E1 17916.55,E2 17916.55} C_VEL
LIN {X 0,Y 368.02,Z 782.534,A -85,B 0,C 180,E1 17913.581,E2 17913.581} C_VEL
LIN {X 0,Y 368.043,Z 783.64,A -85,B 0,C 180,E1 17910.621,E2 17910.621} C_VEL
LIN {X 0,Y 368.035,Z 783.149,A -85,B 0,C 180,E1 17907.663,E2 17907.663} C_VEL
LIN {X 0,Y 368.011,Z 781.189,A -85,B 0,C 180,E1 17904.854,E2 17904.854} C_VEL
LIN {X 0,Y 368.069,Z 777.445,A -85,B 0,C 180,E1 17901.878,E2 17901.878} C_VEL
LIN {X 0,Y 368.282,Z 771.99,A -85,B 0,C 180,E1 17898.885,E2 17898.885} C_VEL
LIN {X 0,Y 368.805,Z 764.701,A -85,B 0,C 180,E1 17895.876,E2 17895.876} C_VEL
LIN {X 0,Y 369.691,Z 755.961,A -85,B 0,C 180,E1 17893.015,E2 17893.015} C_VEL
LIN {X 0,Y 371.059,Z 745.069,A -85,B 0,C 180,E1 17890.121,E2 17890.121} C_VEL
LIN {X 0,Y 372.804,Z 732.852,A -85,B 0,C 180,E1 17887.446,E2 17887.446} C_VEL
LIN {X 0,Y 374.959,Z 718.978,A -85,B 0,C 180,E1 17884.912,E2 17884.912} C_VEL
LIN {X 0,Y 377.339,Z 704.103,A -85,B 0,C 180,E1 17882.629,E2 17882.629} C_VEL
LIN {X 0,Y 379.992,Z 687.829,A -85,B 0,C 180,E1 17880.523,E2 17880.523} C_VEL
LIN {X 0,Y 382.806,Z 670.038,A -85,B 0,C 180,E1 17878.594,E2 17878.594} C_VEL
LIN {X 0,Y 385.753,Z 650.514,A -85,B 0,C 180,E1 17876.844,E2 17876.844} C_VEL
LIN {X 0,Y 388.648,Z 629.964,A -85,B 0,C 180,E1 17875.349,E2 17875.349} C_VEL
LIN {X 0,Y 391.397,Z 608.329,A -85,B 0,C 180,E1 17874.096,E2 17874.096} C_VEL
LIN {X 0,Y 393.844,Z 586.698,A -85,B 0,C 180,E1 17873.145,E2 17873.145} C_VEL
LIN {X 0,Y 395.974,Z 562.993,A -85,B 0,C 180,E1 17872.383,E2 17872.383} C_VEL
LIN {X 0,Y 400.952,Z 503.872,A -85,B 0,C 180,E1 17870.714,E2 17870.714} C_VEL
LIN {X 0,Y 407.588,Z 446.434,A -85,B 0,C 180,E1 17868.947,E2 17868.947} C_VEL
LIN {X 0,Y 416.346,Z 388.579,A -85,B 0,C 180,E1 17867.079,E2 17867.079} C_VEL
LIN {X 0,Y 420.44,Z 365.452,A -85,B 0,C 180,E1 17866.298,E2 17866.298} C_VEL
LIN {X 0,Y 419.53,Z 363.016,A -85,B 0,C 180,E1 17865.446,E2 17865.446} C_VEL
LIN {X 0,Y 418.737,Z 360.955,A -85,B 0,C 180,E1 17864.205,E2 17864.205} C_VEL
LIN {X 0,Y 418.331,Z 361.229,A -85,B 0,C 180,E1 17863.311,E2 17863.311} C_VEL
LIN {X 0,Y 418.348,Z 363.199,A -85,B 0,C 180,E1 17861.913,E2 17861.913} C_VEL
LIN {X 0,Y 419.16,Z 367.683,A -85,B 0,C 180,E1 17860.399,E2 17860.399} C_VEL
LIN {X 0,Y 419.383,Z 369.481,A -85,B 0,C 180,E1 17860.035,E2 17860.035} C_VEL
LIN {X 0,Y 418.006,Z 383.821,A -85,B 0,C 180,E1 17858.993,E2 17858.993} C_VEL
LIN {X 0,Y 406.652,Z 454.241,A -85,B 0,C 180,E1 17856.662,E2 17856.662} C_VEL
LIN {X 0,Y 398.55,Z 518.695,A -85,B 0,C 180,E1 17854.55,E2 17854.55} C_VEL
LIN {X 0,Y 393.19,Z 572.044,A -85,B 0,C 180,E1 17852.828,E2 17852.828} C_VEL
LIN {X 0,Y 390.813,Z 592.528,A -85,B 0,C 180,E1 17851.891,E2 17851.891} C_VEL
LIN {X 0,Y 388.137,Z 612.992,A -85,B 0,C 180,E1 17850.667,E2 17850.667} C_VEL
LIN {X 0,Y 385.32,Z 632.248,A -85,B 0,C 180,E1 17849.198,E2 17849.198} C_VEL
LIN {X 0,Y 382.563,Z 649.759,A -85,B 0,C 180,E1 17847.555,E2 17847.555} C_VEL
LIN {X 0,Y 379.805,Z 666.333,A -85,B 0,C 180,E1 17845.661,E2 17845.661} C_VEL
LIN {X 0,Y 377.138,Z 681.804,A -85,B 0,C 180,E1 17843.515,E2 17843.515} C_VEL
LIN {X 0,Y 374.817,Z 695.181,A -85,B 0,C 180,E1 17841.271,E2 17841.271} C_VEL
LIN {X 0,Y 372.735,Z 707.431,A -85,B 0,C 180,E1 17838.777,E2 17838.777} C_VEL
LIN {X 0,Y 371.118,Z 717.485,A -85,B 0,C 180,E1 17836.271,E2 17836.271} C_VEL
LIN {X 0,Y 369.861,Z 726.123,A -85,B 0,C 180,E1 17833.602,E2 17833.602} C_VEL
LIN {X 0,Y 368.975,Z 733.258,A -85,B 0,C 180,E1 17830.776,E2 17830.776} C_VEL
LIN {X 0,Y 368.446,Z 738.52,A -85,B 0,C 180,E1 17827.955,E2 17827.955} C_VEL
LIN {X 0,Y 368.187,Z 742.055,A -85,B 0,C 180,E1 17825.141,E2 17825.141} C_VEL
LIN {X 0,Y 368.078,Z 743.947,A -85,B 0,C 180,E1 17822.335,E2 17822.335} C_VEL
LIN {X 0,Y 368.051,Z 744.24,A -85,B 0,C 180,E1 17819.532,E2 17819.532} C_VEL
LIN {X 0,Y 368.066,Z 742.931,A -85,B 0,C 180,E1 17816.729,E2 17816.729} C_VEL
LIN {X 0,Y 368.166,Z 740.004,A -85,B 0,C 180,E1 17813.919,E2 17813.919} C_VEL
LIN {X 0,Y 368.438,Z 735.283,A -85,B 0,C 180,E1 17811.052,E2 17811.052} C_VEL
LIN {X 0,Y 368.976,Z 728.947,A -85,B 0,C 180,E1 17808.273,E2 17808.273} C_VEL
LIN {X 0,Y 369.827,Z 721.055,A -85,B 0,C 180,E1 17805.597,E2 17805.597} C_VEL
LIN {X 0,Y 371.003,Z 711.81,A -85,B 0,C 180,E1 17803.078,E2 17803.078} C_VEL
LIN {X 0,Y 372.593,Z 700.493,A -85,B 0,C 180,E1 17800.563,E2 17800.563} C_VEL
LIN {X 0,Y 374.5,Z 687.664,A -85,B 0,C 180,E1 17798.215,E2 17798.215} C_VEL
LIN {X 0,Y 376.673,Z 673.272,A -85,B 0,C 180,E1 17796.037,E2 17796.037} C_VEL
LIN {X 0,Y 378.915,Z 658.124,A -85,B 0,C 180,E1 17794.135,E2 17794.135} C_VEL
LIN {X 0,Y 381.192,Z 641.872,A -85,B 0,C 180,E1 17792.447,E2 17792.447} C_VEL
LIN {X 0,Y 383.414,Z 624.653,A -85,B 0,C 180,E1 17790.984,E2 17790.984} C_VEL
LIN {X 0,Y 385.514,Z 606.259,A -85,B 0,C 180,E1 17789.732,E2 17789.732} C_VEL
LIN {X 0,Y 387.38,Z 586.654,A -85,B 0,C 180,E1 17788.703,E2 17788.703} C_VEL
LIN {X 0,Y 388.941,Z 566.164,A -85,B 0,C 180,E1 17787.931,E2 17787.931} C_VEL
LIN {X 0,Y 390.345,Z 536.46,A -85,B 0,C 180,E1 17787.204,E2 17787.204} C_VEL
LIN {X 0,Y 397.577,Z 377.275,A -85,B 0,C 180,E1 17783.581,E2 17783.581} C_VEL
LIN {X 0,Y 393.441,Z 348.721,A -85,B 0,C 180,E1 17782.369,E2 17782.369} C_VEL
LIN {X 0,Y 388.564,Z 339.103,A -85,B 0,C 180,E1 17781.529,E2 17781.529} C_VEL
LIN {X 0,Y 381.373,Z 319.703,A -85,B 0,C 180,E1 17778.246,E2 17778.246} C_VEL
LIN {X 0,Y 374.161,Z 301.415,A -85,B 0,C 180,E1 17774.87,E2 17774.87} C_VEL
LIN {X 0,Y 369.778,Z 290.655,A -85,B 0,C 180,E1 17772.684,E2 17772.684} C_VEL
LIN {X 0,Y 369.749,Z 290.429,A -85,B 0,C 180,E1 17768.601,E2 17768.601} C_VEL
LIN {X 0,Y 369.743,Z 290.426,A -85,B 0,C 180,E1 17764.416,E2 17764.416} C_VEL
LIN {X 0,Y 369.747,Z 290.411,A -85,B 0,C 180,E1 17760.378,E2 17760.378} C_VEL
LIN {X 0,Y 369.739,Z 290.421,A -85,B 0,C 180,E1 17756.328,E2 17756.328} C_VEL
LIN {X 0,Y 369.744,Z 290.418,A -85,B 0,C 180,E1 17752.248,E2 17752.248} C_VEL
LIN {X 0,Y 369.75,Z 290.681,A -85,B 0,C 180,E1 17751.205,E2 17751.205} C_VEL
LIN {X 0,Y 378.347,Z 311.374,A -85,B 0,C 180,E1 17747.939,E2 17747.939} C_VEL
LIN {X 0,Y 385.096,Z 329.918,A -85,B 0,C 180,E1 17745.281,E2 17745.281} C_VEL
LIN {X 0,Y 388.637,Z 341.241,A -85,B 0,C 180,E1 17743.769,E2 17743.769} C_VEL
LIN {X 0,Y 386.021,Z 382.579,A -85,B 0,C 180,E1 17739.845,E2 17739.845} C_VEL
LIN {X 0,Y 384.433,Z 407.611,A -85,B 0,C 180,E1 17737.475,E2 17737.475} C_VEL
LIN {X 0,Y 383.132,Z 414.289,A -85,B 0,C 180,E1 17736.917,E2 17736.917} C_VEL
LIN {X 0,Y 376.341,Z 432.592,A -85,B 0,C 180,E1 17735.645,E2 17735.645} C_VEL
LIN {X 0,Y 375.3,Z 438.327,A -85,B 0,C 180,E1 17735.151,E2 17735.151} C_VEL
LIN {X 0,Y 372.631,Z 480.345,A -85,B 0,C 180,E1 17731.15,E2 17731.15} C_VEL
LIN {X 0,Y 374.555,Z 499.287,A -85,B 0,C 180,E1 17730.609,E2 17730.609} C_VEL
LIN {X 0,Y 371.744,Z 623.954,A -85,B 0,C 180,E1 17728.133,E2 17728.133} C_VEL
LIN {X 0,Y 371.04,Z 640.012,A -85,B 0,C 180,E1 17727.531,E2 17727.531} C_VEL
LIN {X 0,Y 369.982,Z 655.877,A -85,B 0,C 180,E1 17726.643,E2 17726.643} C_VEL
LIN {X 0,Y 368.737,Z 669.994,A -85,B 0,C 180,E1 17725.57,E2 17725.57} C_VEL
LIN {X 0,Y 367.225,Z 684.313,A -85,B 0,C 180,E1 17724.154,E2 17724.154} C_VEL
LIN {X 0,Y 365.703,Z 697.159,A -85,B 0,C 180,E1 17722.54,E2 17722.54} C_VEL
LIN {X 0,Y 364.22,Z 708.895,A -85,B 0,C 180,E1 17720.681,E2 17720.681} C_VEL
LIN {X 0,Y 362.949,Z 718.813,A -85,B 0,C 180,E1 17718.723,E2 17718.723} C_VEL
LIN {X 0,Y 361.809,Z 727.957,A -85,B 0,C 180,E1 17716.416,E2 17716.416} C_VEL
LIN {X 0,Y 361.014,Z 735.082,A -85,B 0,C 180,E1 17714.088,E2 17714.088} C_VEL
LIN {X 0,Y 360.481,Z 740.708,A -85,B 0,C 180,E1 17711.552,E2 17711.552} C_VEL
LIN {X 0,Y 360.22,Z 744.468,A -85,B 0,C 180,E1 17709.021,E2 17709.021} C_VEL
LIN {X 0,Y 360.115,Z 746.468,A -85,B 0,C 180,E1 17706.385,E2 17706.385} C_VEL
LIN {X 0,Y 360.118,Z 746.707,A -85,B 0,C 180,E1 17703.805,E2 17703.805} C_VEL
LIN {X 0,Y 360.212,Z 745.207,A -85,B 0,C 180,E1 17701.301,E2 17701.301} C_VEL
LIN {X 0,Y 360.482,Z 741.88,A -85,B 0,C 180,E1 17698.683,E2 17698.683} C_VEL
LIN {X 0,Y 360.99,Z 736.788,A -85,B 0,C 180,E1 17696.173,E2 17696.173} C_VEL
LIN {X 0,Y 361.814,Z 729.961,A -85,B 0,C 180,E1 17693.748,E2 17693.748} C_VEL
LIN {X 0,Y 362.929,Z 721.526,A -85,B 0,C 180,E1 17691.483,E2 17691.483} C_VEL
LIN {X 0,Y 364.342,Z 711.321,A -85,B 0,C 180,E1 17689.337,E2 17689.337} C_VEL
LIN {X 0,Y 365.805,Z 700.533,A -85,B 0,C 180,E1 17687.539,E2 17687.539} C_VEL
LIN {X 0,Y 367.422,Z 687.824,A -85,B 0,C 180,E1 17685.844,E2 17685.844} C_VEL
LIN {X 0,Y 368.904,Z 674.932,A -85,B 0,C 180,E1 17684.477,E2 17684.477} C_VEL
LIN {X 0,Y 370.302,Z 660.652,A -85,B 0,C 180,E1 17683.302,E2 17683.302} C_VEL
LIN {X 0,Y 371.494,Z 645.139,A -85,B 0,C 180,E1 17682.341,E2 17682.341} C_VEL
LIN {X 0,Y 372.331,Z 628.571,A -85,B 0,C 180,E1 17681.645,E2 17681.645} C_VEL
LIN {X 0,Y 372.829,Z 609.797,A -85,B 0,C 180,E1 17681.189,E2 17681.189} C_VEL
LIN {X 0,Y 375.331,Z 496.579,A -85,B 0,C 180,E1 17678.943,E2 17678.943} C_VEL
LIN {X 0,Y 373.529,Z 480.228,A -85,B 0,C 180,E1 17678.391,E2 17678.391} C_VEL
LIN {X 0,Y 376.355,Z 437.011,A -85,B 0,C 180,E1 17674.291,E2 17674.291} C_VEL
LIN {X 0,Y 379.094,Z 395.27,A -85,B 0,C 180,E1 17670.346,E2 17670.346} C_VEL
LIN {X 0,Y 381.738,Z 352.371,A -85,B 0,C 180,E1 17666.329,E2 17666.329} C_VEL
LIN {X 0,Y 382.179,Z 342.798,A -85,B 0,C 180,E1 17665.408,E2 17665.408} C_VEL
LIN {X 0,Y 376.531,Z 325.559,A -85,B 0,C 180,E1 17662.977,E2 17662.977} C_VEL
LIN {X 0,Y 370.306,Z 310.03,A -85,B 0,C 180,E1 17660.55,E2 17660.55} C_VEL
LIN {X 0,Y 364.847,Z 298.49,A -85,B 0,C 180,E1 17658.536,E2 17658.536} C_VEL
LIN {X 0,Y 361.863,Z 291.816,A -85,B 0,C 180,E1 17657.28,E2 17657.28} C_VEL
LIN {X 0,Y 361.776,Z 291.421,A -85,B 0,C 180,E1 17656.705,E2 17656.705} C_VEL
LIN {X 0,Y 361.777,Z 291.421,A -85,B 0,C 180,E1 17652.612,E2 17652.612} C_VEL
LIN {X 0,Y 361.775,Z 291.418,A -85,B 0,C 180,E1 17648.424,E2 17648.424} C_VEL
LIN {X 0,Y 361.776,Z 291.417,A -85,B 0,C 180,E1 17644.28,E2 17644.28} C_VEL
LIN {X 0,Y 361.777,Z 291.421,A -85,B 0,C 180,E1 17640.159,E2 17640.159} C_VEL
LIN {X 0,Y 361.777,Z 291.414,A -85,B 0,C 180,E1 17636.039,E2 17636.039} C_VEL
LIN {X 0,Y 361.78,Z 291.42,A -85,B 0,C 180,E1 17631.898,E2 17631.898} C_VEL
LIN {X 0,Y 361.786,Z 291.414,A -85,B 0,C 180,E1 17627.714,E2 17627.714} C_VEL
LIN {X 0,Y 361.79,Z 291.413,A -85,B 0,C 180,E1 17623.627,E2 17623.627} C_VEL
LIN {X 0,Y 361.799,Z 291.42,A -85,B 0,C 180,E1 17619.454,E2 17619.454} C_VEL
LIN {X 0,Y 361.801,Z 291.414,A -85,B 0,C 180,E1 17615.336,E2 17615.336} C_VEL
LIN {X 0,Y 361.818,Z 291.415,A -85,B 0,C 180,E1 17611.08,E2 17611.08} C_VEL
LIN {X 0,Y 361.809,Z 291.418,A -85,B 0,C 180,E1 17606.856,E2 17606.856} C_VEL
LIN {X 0,Y 361.808,Z 291.417,A -85,B 0,C 180,E1 17602.735,E2 17602.735} C_VEL
LIN {X 0,Y 361.853,Z 291.791,A -85,B 0,C 180,E1 17601.399,E2 17601.399} C_VEL
LIN {X 0,Y 370.051,Z 310.673,A -85,B 0,C 180,E1 17597.718,E2 17597.718} C_VEL
LIN {X 0,Y 374.269,Z 320.363,A -85,B 0,C 180,E1 17596.033,E2 17596.033} C_VEL
LIN {X 0,Y 391.264,Z 349.93,A -85,B 0,C 180,E1 17593.176,E2 17593.176} C_VEL
LIN {X 0,Y 396.467,Z 359.906,A -85,B 0,C 180,E1 17592.338,E2 17592.338} C_VEL
LIN {X 0,Y 387.034,Z 557.79,A -85,B 0,C 180,E1 17587.909,E2 17587.909} C_VEL
LIN {X 0,Y 385.672,Z 582.621,A -85,B 0,C 180,E1 17587.271,E2 17587.271} C_VEL
LIN {X 0,Y 383.819,Z 604.013,A -85,B 0,C 180,E1 17586.458,E2 17586.458} C_VEL
LIN {X 0,Y 381.572,Z 624.706,A -85,B 0,C 180,E1 17585.385,E2 17585.385} C_VEL
LIN {X 0,Y 378.957,Z 645.216,A -85,B 0,C 180,E1 17584.008,E2 17584.008} C_VEL
LIN {X 0,Y 376.163,Z 664.59,A -85,B 0,C 180,E1 17582.382,E2 17582.382} C_VEL
LIN {X 0,Y 373.295,Z 682.905,A -85,B 0,C 180,E1 17580.5,E2 17580.5} C_VEL
LIN {X 0,Y 370.468,Z 700.128,A -85,B 0,C 180,E1 17578.357,E2 17578.357} C_VEL
LIN {X 0,Y 367.863,Z 715.674,A -85,B 0,C 180,E1 17576.035,E2 17576.035} C_VEL
LIN {X 0,Y 365.568,Z 729.69,A -85,B 0,C 180,E1 17573.534,E2 17573.534} C_VEL
LIN {X 0,Y 363.692,Z 741.895,A -85,B 0,C 180,E1 17570.938,E2 17570.938} C_VEL
LIN {X 0,Y 362.195,Z 752.719,A -85,B 0,C 180,E1 17568.174,E2 17568.174} C_VEL
LIN {X 0,Y 361.109,Z 762.048,A -85,B 0,C 180,E1 17565.249,E2 17565.249} C_VEL
LIN {X 0,Y 360.45,Z 769.492,A -85,B 0,C 180,E1 17562.331,E2 17562.331} C_VEL
LIN {X 0,Y 360.116,Z 775.518,A -85,B 0,C 180,E1 17559.265,E2 17559.265} C_VEL
LIN {X 0,Y 360.029,Z 779.619,A -85,B 0,C 180,E1 17556.376,E2 17556.376} C_VEL
LIN {X 0,Y 360.031,Z 782.152,A -85,B 0,C 180,E1 17553.501,E2 17553.501} C_VEL
LIN {X 0,Y 360.056,Z 783.184,A -85,B 0,C 180,E1 17550.635,E2 17550.635} C_VEL
LIN {X 0,Y 360.046,Z 782.801,A -85,B 0,C 180,E1 17547.77,E2 17547.77} C_VEL
LIN {X 0,Y 360.019,Z 780.891,A -85,B 0,C 180,E1 17544.9,E2 17544.9} C_VEL
LIN {X 0,Y 360.071,Z 777.255,A -85,B 0,C 180,E1 17541.857,E2 17541.857} C_VEL
LIN {X 0,Y 360.29,Z 771.904,A -85,B 0,C 180,E1 17538.797,E2 17538.797} C_VEL
LIN {X 0,Y 360.802,Z 765.169,A -85,B 0,C 180,E1 17535.884,E2 17535.884} C_VEL
LIN {X 0,Y 361.715,Z 756.614,A -85,B 0,C 180,E1 17532.96,E2 17532.96} C_VEL
LIN {X 0,Y 363.113,Z 746.047,A -85,B 0,C 180,E1 17530.034,E2 17530.034} C_VEL
LIN {X 0,Y 364.945,Z 733.976,A -85,B 0,C 180,E1 17527.274,E2 17527.274} C_VEL
LIN {X 0,Y 367.19,Z 720.436,A -85,B 0,C 180,E1 17524.689,E2 17524.689} C_VEL
LIN {X 0,Y 369.866,Z 704.884,A -85,B 0,C 180,E1 17522.203,E2 17522.203} C_VEL
LIN {X 0,Y 372.777,Z 688.278,A -85,B 0,C 180,E1 17519.983,E2 17519.983} C_VEL
LIN {X 0,Y 375.897,Z 670.021,A -85,B 0,C 180,E1 17517.949,E2 17517.949} C_VEL
LIN {X 0,Y 379.18,Z 649.853,A -85,B 0,C 180,E1 17516.101,E2 17516.101} C_VEL
LIN {X 0,Y 382.324,Z 629.271,A -85,B 0,C 180,E1 17514.573,E2 17514.573} C_VEL
LIN {X 0,Y 385.372,Z 607.362,A -85,B 0,C 180,E1 17513.278,E2 17513.278} C_VEL
LIN {X 0,Y 388.095,Z 585.513,A -85,B 0,C 180,E1 17512.297,E2 17512.297} C_VEL
LIN {X 0,Y 390.531,Z 561.018,A -85,B 0,C 180,E1 17511.491,E2 17511.491} C_VEL
LIN {X 0,Y 396.15,Z 504.027,A -85,B 0,C 180,E1 17509.79,E2 17509.79} C_VEL
LIN {X 0,Y 403.596,Z 448.199,A -85,B 0,C 180,E1 17507.993,E2 17507.993} C_VEL
LIN {X 0,Y 413.32,Z 391.687,A -85,B 0,C 180,E1 17506.113,E2 17506.113} C_VEL
LIN {X 0,Y 417.462,Z 370.843,A -85,B 0,C 180,E1 17505.397,E2 17505.397} C_VEL
LIN {X 0,Y 416.625,Z 368.637,A -85,B 0,C 180,E1 17503.947,E2 17503.947} C_VEL
LIN {X 0,Y 416.23,Z 370.282,A -85,B 0,C 180,E1 17502.352,E2 17502.352} C_VEL
LIN {X 0,Y 416.609,Z 374.396,A -85,B 0,C 180,E1 17500.886,E2 17500.886} C_VEL
LIN {X 0,Y 416.295,Z 377.115,A -85,B 0,C 180,E1 17500.625,E2 17500.625} C_VEL
LIN {X 0,Y 414.994,Z 386.565,A -85,B 0,C 180,E1 17499.964,E2 17499.964} C_VEL
LIN {X 0,Y 402.614,Z 455.585,A -85,B 0,C 180,E1 17497.622,E2 17497.622} C_VEL
LIN {X 0,Y 393.658,Z 518.567,A -85,B 0,C 180,E1 17495.476,E2 17495.476} C_VEL
LIN {X 0,Y 387.47,Z 572.808,A -85,B 0,C 180,E1 17493.641,E2 17493.641} C_VEL
LIN {X 0,Y 384.736,Z 593.941,A -85,B 0,C 180,E1 17492.632,E2 17492.632} C_VEL
LIN {X 0,Y 381.83,Z 613.98,A -85,B 0,C 180,E1 17491.386,E2 17491.386} C_VEL
LIN {X 0,Y 378.704,Z 633.508,A -85,B 0,C 180,E1 17489.846,E2 17489.846} C_VEL
LIN {X 0,Y 375.638,Z 651.411,A -85,B 0,C 180,E1 17488.107,E2 17488.107} C_VEL
LIN {X 0,Y 372.601,Z 668.27,A -85,B 0,C 180,E1 17486.109,E2 17486.109} C_VEL
LIN {X 0,Y 369.779,Z 683.433,A -85,B 0,C 180,E1 17483.928,E2 17483.928} C_VEL
LIN {X 0,Y 367.393,Z 696.148,A -85,B 0,C 180,E1 17481.723,E2 17481.723} C_VEL
LIN {X 0,Y 365.287,Z 707.58,A -85,B 0,C 180,E1 17479.341,E2 17479.341} C_VEL
LIN {X 0,Y 363.518,Z 717.679,A -85,B 0,C 180,E1 17476.786,E2 17476.786} C_VEL
LIN {X 0,Y 362.121,Z 726.367,A -85,B 0,C 180,E1 17474.062,E2 17474.062} C_VEL
LIN {X 0,Y 361.126,Z 733.552,A -85,B 0,C 180,E1 17471.175,E2 17471.175} C_VEL
LIN {X 0,Y 360.532,Z 738.865,A -85,B 0,C 180,E1 17468.291,E2 17468.291} C_VEL
LIN {X 0,Y 360.229,Z 742.445,A -85,B 0,C 180,E1 17465.415,E2 17465.415} C_VEL
LIN {X 0,Y 360.095,Z 744.439,A -85,B 0,C 180,E1 17462.386,E2 17462.386} C_VEL
LIN {X 0,Y 360.063,Z 744.673,A -85,B 0,C 180,E1 17459.522,E2 17459.522} C_VEL
LIN {X 0,Y 360.078,Z 743.299,A -85,B 0,C 180,E1 17456.656,E2 17456.656} C_VEL
LIN {X 0,Y 360.185,Z 740.297,A -85,B 0,C 180,E1 17453.784,E2 17453.784} C_VEL
LIN {X 0,Y 360.473,Z 735.589,A -85,B 0,C 180,E1 17450.903,E2 17450.903} C_VEL
LIN {X 0,Y 361.018,Z 729.481,A -85,B 0,C 180,E1 17448.173,E2 17448.173} C_VEL
LIN {X 0,Y 361.907,Z 721.59,A -85,B 0,C 180,E1 17445.438,E2 17445.438} C_VEL
LIN {X 0,Y 363.22,Z 711.678,A -85,B 0,C 180,E1 17442.704,E2 17442.704} C_VEL
LIN {X 0,Y 364.906,Z 700.221,A -85,B 0,C 180,E1 17440.137,E2 17440.137} C_VEL
LIN {X 0,Y 366.92,Z 687.23,A -85,B 0,C 180,E1 17437.741,E2 17437.741} C_VEL
LIN {X 0,Y 369.206,Z 672.655,A -85,B 0,C 180,E1 17435.521,E2 17435.521} C_VEL
LIN {X 0,Y 371.695,Z 656.362,A -85,B 0,C 180,E1 17433.477,E2 17433.477} C_VEL
LIN {X 0,Y 374.101,Z 639.723,A -85,B 0,C 180,E1 17431.766,E2 17431.766} C_VEL
LIN {X 0,Y 376.392,Z 622.31,A -85,B 0,C 180,E1 17430.304,E2 17430.304} C_VEL
LIN {X 0,Y 378.516,Z 604.11,A -85,B 0,C 180,E1 17429.084,E2 17429.084} C_VEL
LIN {X 0,Y 380.423,Z 584.401,A -85,B 0,C 180,E1 17428.065,E2 17428.065} C_VEL
LIN {X 0,Y 381.947,Z 564.641,A -85,B 0,C 180,E1 17427.332,E2 17427.332} C_VEL
LIN {X 0,Y 384.109,Z 518.749,A -85,B 0,C 180,E1 17426.225,E2 17426.225} C_VEL
LIN {X 0,Y 390.905,Z 378.386,A -85,B 0,C 180,E1 17422.945,E2 17422.945} C_VEL
LIN {X 0,Y 387.233,Z 352.342,A -85,B 0,C 180,E1 17421.807,E2 17421.807} C_VEL
LIN {X 0,Y 380.321,Z 338.936,A -85,B 0,C 180,E1 17420.619,E2 17420.619} C_VEL
LIN {X 0,Y 372.972,Z 319.156,A -85,B 0,C 180,E1 17417.157,E2 17417.157} C_VEL
LIN {X 0,Y 365.795,Z 301.475,A -85,B 0,C 180,E1 17413.754,E2 17413.754} C_VEL
LIN {X 0,Y 361.828,Z 291.608,A -85,B 0,C 180,E1 17411.679,E2 17411.679} C_VEL
LIN {X 0,Y 361.805,Z 291.418,A -85,B 0,C 180,E1 17407.52,E2 17407.52} C_VEL
LIN {X 0,Y 361.803,Z 291.417,A -85,B 0,C 180,E1 17403.365,E2 17403.365} C_VEL
LIN {X 0,Y 361.793,Z 291.394,A -85,B 0,C 180,E1 17399.287,E2 17399.287} C_VEL
LIN {X 0,Y 361.781,Z 291.399,A -85,B 0,C 180,E1 17395.191,E2 17395.191} C_VEL
LIN {X 0,Y 361.849,Z 291.658,A -85,B 0,C 180,E1 17392.118,E2 17392.118} C_VEL
LIN {X 0,Y 364.914,Z 298.892,A -85,B 0,C 180,E1 17390.877,E2 17390.877} C_VEL
LIN {X 0,Y 372.715,Z 317.86,A -85,B 0,C 180,E1 17387.89,E2 17387.89} C_VEL
LIN {X 0,Y 379.259,Z 336.41,A -85,B 0,C 180,E1 17385.222,E2 17385.222} C_VEL
LIN {X 0,Y 381.599,Z 344.037,A -85,B 0,C 180,E1 17384.192,E2 17384.192} C_VEL
LIN {X 0,Y 378.865,Z 384.794,A -85,B 0,C 180,E1 17380.278,E2 17380.278} C_VEL
LIN {X 0,Y 376.074,Z 426.012,A -85,B 0,C 180,E1 17376.336,E2 17376.336} C_VEL
LIN {X 0,Y 375.3,Z 438.327,A -85,B 0,C 180,E1 17375.151,E2 17375.151} C_VEL
LIN {X 0,Y 373.99,Z 445.018,A -85,B 0,C 180,E1 17374.584,E2 17374.584} C_VEL
LIN {X 0,Y 367.132,Z 463.306,A -85,B 0,C 180,E1 17373.284,E2 17373.284} C_VEL
LIN {X 0,Y 366.041,Z 469.044,A -85,B 0,C 180,E1 17372.779,E2 17372.779} C_VEL
LIN {X 0,Y 365.34,Z 480.845,A -85,B 0,C 180,E1 17371.678,E2 17371.678} C_VEL
LIN {X 0,Y 367.274,Z 500.091,A -85,B 0,C 180,E1 17371.113,E2 17371.113} C_VEL
LIN {X 0,Y 364.343,Z 624.371,A -85,B 0,C 180,E1 17368.601,E2 17368.601} C_VEL
LIN {X 0,Y 363.607,Z 640.39,A -85,B 0,C 180,E1 17367.989,E2 17367.989} C_VEL
LIN {X 0,Y 362.484,Z 656.498,A -85,B 0,C 180,E1 17367.069,E2 17367.069} C_VEL
LIN {X 0,Y 361.159,Z 670.777,A -85,B 0,C 180,E1 17365.954,E2 17365.954} C_VEL
LIN {X 0,Y 359.596,Z 684.917,A -85,B 0,C 180,E1 17364.523,E2 17364.523} C_VEL
LIN {X 0,Y 358.065,Z 697.249,A -85,B 0,C 180,E1 17362.944,E2 17362.944} C_VEL
LIN {X 0,Y 356.414,Z 709.709,A -85,B 0,C 180,E1 17360.927,E2 17360.927} C_VEL
LIN {X 0,Y 355.108,Z 719.37,A -85,B 0,C 180,E1 17358.964,E2 17358.964} C_VEL
LIN {X 0,Y 353.909,Z 728.488,A -85,B 0,C 180,E1 17356.607,E2 17356.607} C_VEL
LIN {X 0,Y 353.071,Z 735.573,A -85,B 0,C 180,E1 17354.227,E2 17354.227} C_VEL
LIN {X 0,Y 352.513,Z 741.144,A -85,B 0,C 180,E1 17351.651,E2 17351.651} C_VEL
LIN {X 0,Y 352.233,Z 744.901,A -85,B 0,C 180,E1 17349.045,E2 17349.045} C_VEL
LIN {X 0,Y 352.125,Z 746.856,A -85,B 0,C 180,E1 17346.401,E2 17346.401} C_VEL
LIN {X 0,Y 352.13,Z 747.086,A -85,B 0,C 180,E1 17343.71,E2 17343.71} C_VEL
LIN {X 0,Y 352.235,Z 745.556,A -85,B 0,C 180,E1 17341.149,E2 17341.149} C_VEL
LIN {X 0,Y 352.521,Z 742.31,A -85,B 0,C 180,E1 17338.544,E2 17338.544} C_VEL
LIN {X 0,Y 353.041,Z 737.486,A -85,B 0,C 180,E1 17336.081,E2 17336.081} C_VEL
LIN {X 0,Y 353.901,Z 730.768,A -85,B 0,C 180,E1 17333.611,E2 17333.611} C_VEL
LIN {X 0,Y 355.064,Z 722.531,A -85,B 0,C 180,E1 17331.31,E2 17331.31} C_VEL
LIN {X 0,Y 356.577,Z 712.182,A -85,B 0,C 180,E1 17329.063,E2 17329.063} C_VEL
LIN {X 0,Y 358.152,Z 701.269,A -85,B 0,C 180,E1 17327.187,E2 17327.187} C_VEL
LIN {X 0,Y 359.962,Z 687.793,A -85,B 0,C 180,E1 17325.355,E2 17325.355} C_VEL
LIN {X 0,Y 361.603,Z 674.011,A -85,B 0,C 180,E1 17323.893,E2 17323.893} C_VEL
LIN {X 0,Y 363.109,Z 659.138,A -85,B 0,C 180,E1 17322.678,E2 17322.678} C_VEL
LIN {X 0,Y 364.287,Z 643.643,A -85,B 0,C 180,E1 17321.746,E2 17321.746} C_VEL
LIN {X 0,Y 365.139,Z 626.953,A -85,B 0,C 180,E1 17321.063,E2 17321.063} C_VEL
LIN {X 0,Y 365.879,Z 597.165,A -85,B 0,C 180,E1 17320.406,E2 17320.406} C_VEL
LIN {X 0,Y 368.221,Z 497.455,A -85,B 0,C 180,E1 17318.388,E2 17318.388} C_VEL
LIN {X 0,Y 366.373,Z 481.041,A -85,B 0,C 180,E1 17317.836,E2 17317.836} C_VEL
LIN {X 0,Y 369.311,Z 437.955,A -85,B 0,C 180,E1 17313.712,E2 17313.712} C_VEL
LIN {X 0,Y 372.235,Z 396.103,A -85,B 0,C 180,E1 17309.709,E2 17309.709} C_VEL
LIN {X 0,Y 374.913,Z 355.379,A -85,B 0,C 180,E1 17305.852,E2 17305.852} C_VEL
LIN {X 0,Y 375.452,Z 346.139,A -85,B 0,C 180,E1 17304.968,E2 17304.968} C_VEL
LIN {X 0,Y 370.078,Z 329.501,A -85,B 0,C 180,E1 17302.561,E2 17302.561} C_VEL
LIN {X 0,Y 363.906,Z 314.09,A -85,B 0,C 180,E1 17300.088,E2 17300.088} C_VEL
LIN {X 0,Y 357.873,Z 300.913,A -85,B 0,C 180,E1 17297.731,E2 17297.731} C_VEL
LIN {X 0,Y 355.495,Z 296.371,A -85,B 0,C 180,E1 17296.84,E2 17296.84} C_VEL
LIN {X 0,Y 353.908,Z 292.857,A -85,B 0,C 180,E1 17296.12,E2 17296.12} C_VEL
LIN {X 0,Y 353.868,Z 292.394,A -85,B 0,C 180,E1 17295.537,E2 17295.537} C_VEL
LIN {X 0,Y 353.866,Z 292.409,A -85,B 0,C 180,E1 17291.358,E2 17291.358} C_VEL
LIN {X 0,Y 353.871,Z 292.405,A -85,B 0,C 180,E1 17287.142,E2 17287.142} C_VEL
LIN {X 0,Y 353.854,Z 292.409,A -85,B 0,C 180,E1 17282.916,E2 17282.916} C_VEL
LIN {X 0,Y 353.856,Z 292.401,A -85,B 0,C 180,E1 17278.867,E2 17278.867} C_VEL
LIN {X 0,Y 353.849,Z 292.408,A -85,B 0,C 180,E1 17274.65,E2 17274.65} C_VEL
LIN {X 0,Y 353.847,Z 292.401,A -85,B 0,C 180,E1 17270.568,E2 17270.568} C_VEL
LIN {X 0,Y 353.844,Z 292.407,A -85,B 0,C 180,E1 17266.409,E2 17266.409} C_VEL
LIN {X 0,Y 353.844,Z 292.409,A -85,B 0,C 180,E1 17262.217,E2 17262.217} C_VEL
LIN {X 0,Y 353.839,Z 292.402,A -85,B 0,C 180,E1 17257.925,E2 17257.925} C_VEL
LIN {X 0,Y 353.845,Z 292.41,A -85,B 0,C 180,E1 17253.845,E2 17253.845} C_VEL
LIN {X 0,Y 353.847,Z 292.405,A -85,B 0,C 180,E1 17249.804,E2 17249.804} C_VEL
LIN {X 0,Y 353.85,Z 292.405,A -85,B 0,C 180,E1 17245.589,E2 17245.589} C_VEL
LIN {X 0,Y 353.897,Z 292.66,A -85,B 0,C 180,E1 17242.505,E2 17242.505} C_VEL
LIN {X 0,Y 357.045,Z 299.971,A -85,B 0,C 180,E1 17240.944,E2 17240.944} C_VEL
LIN {X 0,Y 365.164,Z 318.697,A -85,B 0,C 180,E1 17237.338,E2 17237.338} C_VEL
LIN {X 0,Y 366.884,Z 322.019,A -85,B 0,C 180,E1 17236.894,E2 17236.894} C_VEL
LIN {X 0,Y 382.509,Z 349.027,A -85,B 0,C 180,E1 17234.177,E2 17234.177} C_VEL
LIN {X 0,Y 389.851,Z 362.656,A -85,B 0,C 180,E1 17232.964,E2 17232.964} C_VEL
LIN {X 0,Y 379.031,Z 577.128,A -85,B 0,C 180,E1 17228.013,E2 17228.013} C_VEL
LIN {X 0,Y 377.266,Z 598.585,A -85,B 0,C 180,E1 17227.252,E2 17227.252} C_VEL
LIN {X 0,Y 375.037,Z 619.279,A -85,B 0,C 180,E1 17226.239,E2 17226.239} C_VEL
LIN {X 0,Y 372.468,Z 639.496,A -85,B 0,C 180,E1 17224.946,E2 17224.946} C_VEL
LIN {X 0,Y 369.666,Z 658.814,A -85,B 0,C 180,E1 17223.393,E2 17223.393} C_VEL
LIN {X 0,Y 366.714,Z 677.354,A -85,B 0,C 180,E1 17221.565,E2 17221.565} C_VEL
LIN {X 0,Y 363.865,Z 694.194,A -85,B 0,C 180,E1 17219.552,E2 17219.552} C_VEL
LIN {X 0,Y 361.19,Z 709.59,A -85,B 0,C 180,E1 17217.354,E2 17217.354} C_VEL
LIN {X 0,Y 358.686,Z 724.094,A -85,B 0,C 180,E1 17214.891,E2 17214.891} C_VEL
LIN {X 0,Y 356.53,Z 737.136,A -85,B 0,C 180,E1 17212.245,E2 17212.245} C_VEL
LIN {X 0,Y 354.787,Z 748.722,A -85,B 0,C 180,E1 17209.421,E2 17209.421} C_VEL
LIN {X 0,Y 353.51,Z 758.583,A -85,B 0,C 180,E1 17206.502,E2 17206.502} C_VEL
LIN {X 0,Y 352.651,Z 766.912,A -85,B 0,C 180,E1 17203.442,E2 17203.442} C_VEL
LIN {X 0,Y 352.202,Z 773.508,A -85,B 0,C 180,E1 17200.301,E2 17200.301} C_VEL
LIN {X 0,Y 352.042,Z 778.044,A -85,B 0,C 180,E1 17197.341,E2 17197.341} C_VEL
LIN {X 0,Y 352.043,Z 781.185,A -85,B 0,C 180,E1 17194.233,E2 17194.233} C_VEL
LIN {X 0,Y 352.064,Z 782.659,A -85,B 0,C 180,E1 17191.3,E2 17191.3} C_VEL
LIN {X 0,Y 352.063,Z 782.558,A -85,B 0,C 180,E1 17188.371,E2 17188.371} C_VEL
LIN {X 0,Y 352.03,Z 780.87,A -85,B 0,C 180,E1 17185.274,E2 17185.274} C_VEL
LIN {X 0,Y 352.059,Z 777.546,A -85,B 0,C 180,E1 17182.163,E2 17182.163} C_VEL
LIN {X 0,Y 352.265,Z 772.518,A -85,B 0,C 180,E1 17179.036,E2 17179.036} C_VEL
LIN {X 0,Y 352.8,Z 765.61,A -85,B 0,C 180,E1 17175.892,E2 17175.892} C_VEL
LIN {X 0,Y 353.738,Z 757.245,A -85,B 0,C 180,E1 17172.903,E2 17172.903} C_VEL
LIN {X 0,Y 355.188,Z 746.947,A -85,B 0,C 180,E1 17169.912,E2 17169.912} C_VEL
LIN {X 0,Y 357.225,Z 734.416,A -85,B 0,C 180,E1 17166.929,E2 17166.929} C_VEL
LIN {X 0,Y 359.635,Z 720.906,A -85,B 0,C 180,E1 17164.261,E2 17164.261} C_VEL
LIN {X 0,Y 362.434,Z 705.823,A -85,B 0,C 180,E1 17161.761,E2 17161.761} C_VEL
LIN {X 0,Y 365.622,Z 688.919,A -85,B 0,C 180,E1 17159.425,E2 17159.425} C_VEL
LIN {X 0,Y 368.931,Z 671.004,A -85,B 0,C 180,E1 17157.361,E2 17157.361} C_VEL
LIN {X 0,Y 372.339,Z 651.793,A -85,B 0,C 180,E1 17155.527,E2 17155.527} C_VEL
LIN {X 0,Y 375.847,Z 630.868,A -85,B 0,C 180,E1 17153.901,E2 17153.901} C_VEL
LIN {X 0,Y 379.16,Z 609.366,A -85,B 0,C 180,E1 17152.565,E2 17152.565} C_VEL
LIN {X 0,Y 382.265,Z 587.239,A -85,B 0,C 180,E1 17151.51,E2 17151.51} C_VEL
LIN {X 0,Y 385.075,Z 563.095,A -85,B 0,C 180,E1 17150.656,E2 17150.656} C_VEL
LIN {X 0,Y 391.254,Z 508.421,A -85,B 0,C 180,E1 17148.945,E2 17148.945} C_VEL
LIN {X 0,Y 399.432,Z 454.052,A -85,B 0,C 180,E1 17147.13,E2 17147.13} C_VEL
LIN {X 0,Y 409.983,Z 399.107,A -85,B 0,C 180,E1 17145.258,E2 17145.258} C_VEL
LIN {X 0,Y 414.784,Z 377.197,A -85,B 0,C 180,E1 17144.501,E2 17144.501} C_VEL
LIN {X 0,Y 414.542,Z 376.403,A -85,B 0,C 180,E1 17143.807,E2 17143.807} C_VEL
LIN {X 0,Y 414.117,Z 378.19,A -85,B 0,C 180,E1 17142.431,E2 17142.431} C_VEL
LIN {X 0,Y 414.089,Z 380.818,A -85,B 0,C 180,E1 17141.555,E2 17141.555} C_VEL
LIN {X 0,Y 412.662,Z 388.813,A -85,B 0,C 180,E1 17140.985,E2 17140.985} C_VEL
LIN {X 0,Y 398.922,Z 457.859,A -85,B 0,C 180,E1 17138.598,E2 17138.598} C_VEL
LIN {X 0,Y 388.944,Z 520.401,A -85,B 0,C 180,E1 17136.395,E2 17136.395} C_VEL
LIN {X 0,Y 382.044,Z 573.666,A -85,B 0,C 180,E1 17134.507,E2 17134.507} C_VEL
LIN {X 0,Y 378.992,Z 594.737,A -85,B 0,C 180,E1 17133.462,E2 17133.462} C_VEL
LIN {X 0,Y 375.73,Z 615.001,A -85,B 0,C 180,E1 17132.155,E2 17132.155} C_VEL
LIN {X 0,Y 372.349,Z 634.296,A -85,B 0,C 180,E1 17130.587,E2 17130.587} C_VEL
LIN {X 0,Y 368.925,Z 652.617,A -85,B 0,C 180,E1 17128.754,E2 17128.754} C_VEL
LIN {X 0,Y 365.683,Z 669.205,A -85,B 0,C 180,E1 17126.731,E2 17126.731} C_VEL
LIN {X 0,Y 362.675,Z 684.156,A -85,B 0,C 180,E1 17124.523,E2 17124.523} C_VEL
LIN {X 0,Y 360.016,Z 697.247,A -85,B 0,C 180,E1 17122.191,E2 17122.191} C_VEL
LIN {X 0,Y 357.627,Z 709.237,A -85,B 0,C 180,E1 17119.602,E2 17119.602} C_VEL
LIN {X 0,Y 355.652,Z 719.675,A -85,B 0,C 180,E1 17116.832,E2 17116.832} C_VEL
LIN {X 0,Y 354.138,Z 728.499,A -85,B 0,C 180,E1 17113.885,E2 17113.885} C_VEL
LIN {X 0,Y 353.133,Z 735.287,A -85,B 0,C 180,E1 17110.935,E2 17110.935} C_VEL
LIN {X 0,Y 352.533,Z 740.238,A -85,B 0,C 180,E1 17107.988,E2 17107.988} C_VEL
LIN {X 0,Y 352.221,Z 743.615,A -85,B 0,C 180,E1 17104.885,E2 17104.885} C_VEL
LIN {X 0,Y 352.102,Z 745.165,A -85,B 0,C 180,E1 17101.789,E2 17101.789} C_VEL
LIN {X 0,Y 352.078,Z 744.964,A -85,B 0,C 180,E1 17098.86,E2 17098.86} C_VEL
LIN {X 0,Y 352.101,Z 743.142,A -85,B 0,C 180,E1 17095.928,E2 17095.928} C_VEL
LIN {X 0,Y 352.254,Z 739.671,A -85,B 0,C 180,E1 17092.989,E2 17092.989} C_VEL
LIN {X 0,Y 352.635,Z 734.466,A -85,B 0,C 180,E1 17090.039,E2 17090.039} C_VEL
LIN {X 0,Y 353.289,Z 727.831,A -85,B 0,C 180,E1 17087.246,E2 17087.246} C_VEL
LIN {X 0,Y 354.339,Z 719.363,A -85,B 0,C 180,E1 17084.45,E2 17084.45} C_VEL
LIN {X 0,Y 355.767,Z 709.37,A -85,B 0,C 180,E1 17081.795,E2 17081.795} C_VEL
LIN {X 0,Y 357.628,Z 697.449,A -85,B 0,C 180,E1 17079.202,E2 17079.202} C_VEL
LIN {X 0,Y 359.767,Z 684.297,A -85,B 0,C 180,E1 17076.842,E2 17076.842} C_VEL
LIN {X 0,Y 362.151,Z 669.647,A -85,B 0,C 180,E1 17074.663,E2 17074.663} C_VEL
LIN {X 0,Y 364.723,Z 653.29,A -85,B 0,C 180,E1 17072.653,E2 17072.653} C_VEL
LIN {X 0,Y 367.283,Z 635.924,A -85,B 0,C 180,E1 17070.913,E2 17070.913} C_VEL
LIN {X 0,Y 369.705,Z 617.67,A -85,B 0,C 180,E1 17069.439,E2 17069.439} C_VEL
LIN {X 0,Y 371.868,Z 598.902,A -85,B 0,C 180,E1 17068.242,E2 17068.242} C_VEL
LIN {X 0,Y 373.752,Z 579.176,A -85,B 0,C 180,E1 17067.289,E2 17067.289} C_VEL
LIN {X 0,Y 375.216,Z 558.965,A -85,B 0,C 180,E1 17066.602,E2 17066.602} C_VEL
LIN {X 0,Y 384.268,Z 379.693,A -85,B 0,C 180,E1 17062.304,E2 17062.304} C_VEL
LIN {X 0,Y 380.901,Z 355.727,A -85,B 0,C 180,E1 17061.227,E2 17061.227} C_VEL
LIN {X 0,Y 372.105,Z 338.803,A -85,B 0,C 180,E1 17059.672,E2 17059.672} C_VEL
LIN {X 0,Y 364.897,Z 319.706,A -85,B 0,C 180,E1 17056.223,E2 17056.223} C_VEL
LIN {X 0,Y 358.197,Z 303.093,A -85,B 0,C 180,E1 17052.931,E2 17052.931} C_VEL
LIN {X 0,Y 353.898,Z 292.602,A -85,B 0,C 180,E1 17050.654,E2 17050.654} C_VEL
LIN {X 0,Y 353.864,Z 292.405,A -85,B 0,C 180,E1 17046.599,E2 17046.599} C_VEL
LIN {X 0,Y 353.868,Z 292.405,A -85,B 0,C 180,E1 17042.345,E2 17042.345} C_VEL
LIN {X 0,Y 353.878,Z 292.389,A -85,B 0,C 180,E1 17038.156,E2 17038.156} C_VEL
LIN {X 0,Y 353.868,Z 292.392,A -85,B 0,C 180,E1 17033.833,E2 17033.833} C_VEL
LIN {X 0,Y 353.881,Z 292.683,A -85,B 0,C 180,E1 17033.082,E2 17033.082} C_VEL
LIN {X 0,Y 355.345,Z 296.146,A -85,B 0,C 180,E1 17032.432,E2 17032.432} C_VEL
LIN {X 0,Y 363,Z 313.908,A -85,B 0,C 180,E1 17029.47,E2 17029.47} C_VEL
LIN {X 0,Y 369.965,Z 332.505,A -85,B 0,C 180,E1 17026.648,E2 17026.648} C_VEL
LIN {X 0,Y 374.563,Z 347.008,A -85,B 0,C 180,E1 17024.613,E2 17024.613} C_VEL
LIN {X 0,Y 371.681,Z 388.244,A -85,B 0,C 180,E1 17020.62,E2 17020.62} C_VEL
LIN {X 0,Y 368.71,Z 429.481,A -85,B 0,C 180,E1 17016.62,E2 17016.62} C_VEL
LIN {X 0,Y 366.041,Z 469.044,A -85,B 0,C 180,E1 17012.779,E2 17012.779} C_VEL
LIN {X 0,Y 364.887,Z 473.69,A -85,B 0,C 180,E1 17012.432,E2 17012.432} C_VEL
LIN {X 0,Y 360.9,Z 482.615,A -85,B 0,C 180,E1 17012.12,E2 17012.12} C_VEL
LIN {X 0,Y 359.261,Z 488.42,A -85,B 0,C 180,E1 17011.992,E2 17011.992} C_VEL
LIN {X 0,Y 359.22,Z 491.389,A -85,B 0,C 180,E1 17011.911,E2 17011.911} C_VEL
LIN {X 0,Y 360.012,Z 501.251,A -85,B 0,C 180,E1 17011.63,E2 17011.63} C_VEL
LIN {X 0,Y 356.963,Z 624.676,A -85,B 0,C 180,E1 17009.089,E2 17009.089} C_VEL
LIN {X 0,Y 356.194,Z 640.757,A -85,B 0,C 180,E1 17008.464,E2 17008.464} C_VEL
LIN {X 0,Y 355.087,Z 656.045,A -85,B 0,C 180,E1 17007.581,E2 17007.581} C_VEL
LIN {X 0,Y 353.694,Z 670.658,A -85,B 0,C 180,E1 17006.436,E2 17006.436} C_VEL
LIN {X 0,Y 352.026,Z 685.133,A -85,B 0,C 180,E1 17004.95,E2 17004.95} C_VEL
LIN {X 0,Y 350.364,Z 697.92,A -85,B 0,C 180,E1 17003.278,E2 17003.278} C_VEL
LIN {X 0,Y 348.671,Z 710.11,A -85,B 0,C 180,E1 17001.26,E2 17001.26} C_VEL
LIN {X 0,Y 347.272,Z 719.928,A -85,B 0,C 180,E1 16999.216,E2 16999.216} C_VEL
LIN {X 0,Y 346.014,Z 729.02,A -85,B 0,C 180,E1 16996.806,E2 16996.806} C_VEL
LIN {X 0,Y 345.13,Z 736.064,A -85,B 0,C 180,E1 16994.372,E2 16994.372} C_VEL
LIN {X 0,Y 344.524,Z 741.813,A -85,B 0,C 180,E1 16991.625,E2 16991.625} C_VEL
LIN {X 0,Y 344.246,Z 745.333,A -85,B 0,C 180,E1 16989.071,E2 16989.071} C_VEL
LIN {X 0,Y 344.133,Z 747.32,A -85,B 0,C 180,E1 16986.238,E2 16986.238} C_VEL
LIN {X 0,Y 344.142,Z 747.461,A -85,B 0,C 180,E1 16983.61,E2 16983.61} C_VEL
LIN {X 0,Y 344.275,Z 745.73,A -85,B 0,C 180,E1 16980.799,E2 16980.799} C_VEL
LIN {X 0,Y 344.607,Z 742.318,A -85,B 0,C 180,E1 16978.128,E2 16978.128} C_VEL
LIN {X 0,Y 345.259,Z 736.861,A -85,B 0,C 180,E1 16975.419,E2 16975.419} C_VEL
LIN {X 0,Y 346.168,Z 730.414,A -85,B 0,C 180,E1 16973.077,E2 16973.077} C_VEL
LIN {X 0,Y 347.447,Z 721.905,A -85,B 0,C 180,E1 16970.724,E2 16970.724} C_VEL
LIN {X 0,Y 349.057,Z 711.622,A -85,B 0,C 180,E1 16968.49,E2 16968.49} C_VEL
LIN {X 0,Y 350.826,Z 699.81,A -85,B 0,C 180,E1 16966.483,E2 16966.483} C_VEL
LIN {X 0,Y 352.53,Z 687.765,A -85,B 0,C 180,E1 16964.845,E2 16964.845} C_VEL
LIN {X 0,Y 354.266,Z 673.752,A -85,B 0,C 180,E1 16963.348,E2 16963.348} C_VEL
LIN {X 0,Y 355.842,Z 658.826,A -85,B 0,C 180,E1 16962.119,E2 16962.119} C_VEL
LIN {X 0,Y 357.082,Z 642.927,A -85,B 0,C 180,E1 16961.166,E2 16961.166} C_VEL
LIN {X 0,Y 357.937,Z 626.53,A -85,B 0,C 180,E1 16960.499,E2 16960.499} C_VEL
LIN {X 0,Y 359.191,Z 577.723,A -85,B 0,C 180,E1 16959.448,E2 16959.448} C_VEL
LIN {X 0,Y 361.15,Z 498.272,A -85,B 0,C 180,E1 16957.806,E2 16957.806} C_VEL
LIN {X 0,Y 359.27,Z 481.145,A -85,B 0,C 180,E1 16957.202,E2 16957.202} C_VEL
LIN {X 0,Y 362.404,Z 437.841,A -85,B 0,C 180,E1 16952.999,E2 16952.999} C_VEL
LIN {X 0,Y 365.258,Z 398.895,A -85,B 0,C 180,E1 16949.242,E2 16949.242} C_VEL
LIN {X 0,Y 368.005,Z 360.056,A -85,B 0,C 180,E1 16945.518,E2 16945.518} C_VEL
LIN {X 0,Y 368.62,Z 349.005,A -85,B 0,C 180,E1 16944.435,E2 16944.435} C_VEL
LIN {X 0,Y 363.275,Z 332.476,A -85,B 0,C 180,E1 16941.983,E2 16941.983} C_VEL
LIN {X 0,Y 357.268,Z 317.255,A -85,B 0,C 180,E1 16939.454,E2 16939.454} C_VEL
LIN {X 0,Y 350.123,Z 302.104,A -85,B 0,C 180,E1 16936.594,E2 16936.594} C_VEL
LIN {X 0,Y 347.358,Z 297.043,A -85,B 0,C 180,E1 16935.528,E2 16935.528} C_VEL
LIN {X 0,Y 345.947,Z 293.7,A -85,B 0,C 180,E1 16934.778,E2 16934.778} C_VEL
LIN {X 0,Y 345.917,Z 293.398,A -85,B 0,C 180,E1 16933.03,E2 16933.03} C_VEL
LIN {X 0,Y 345.908,Z 293.395,A -85,B 0,C 180,E1 16928.813,E2 16928.813} C_VEL
LIN {X 0,Y 345.904,Z 293.396,A -85,B 0,C 180,E1 16924.643,E2 16924.643} C_VEL
LIN {X 0,Y 345.899,Z 293.399,A -85,B 0,C 180,E1 16920.332,E2 16920.332} C_VEL
LIN {X 0,Y 345.901,Z 293.392,A -85,B 0,C 180,E1 16916.023,E2 16916.023} C_VEL
LIN {X 0,Y 345.904,Z 293.398,A -85,B 0,C 180,E1 16911.858,E2 16911.858} C_VEL
LIN {X 0,Y 345.911,Z 293.391,A -85,B 0,C 180,E1 16907.65,E2 16907.65} C_VEL
LIN {X 0,Y 345.917,Z 293.39,A -85,B 0,C 180,E1 16903.545,E2 16903.545} C_VEL
LIN {X 0,Y 345.926,Z 293.396,A -85,B 0,C 180,E1 16899.353,E2 16899.353} C_VEL
LIN {X 0,Y 345.928,Z 293.39,A -85,B 0,C 180,E1 16895.166,E2 16895.166} C_VEL
LIN {X 0,Y 345.94,Z 293.391,A -85,B 0,C 180,E1 16890.951,E2 16890.951} C_VEL
LIN {X 0,Y 345.926,Z 293.395,A -85,B 0,C 180,E1 16886.645,E2 16886.645} C_VEL
LIN {X 0,Y 345.947,Z 293.653,A -85,B 0,C 180,E1 16883.623,E2 16883.623} C_VEL
LIN {X 0,Y 349.101,Z 300.999,A -85,B 0,C 180,E1 16881.992,E2 16881.992} C_VEL
LIN {X 0,Y 356.998,Z 319.001,A -85,B 0,C 180,E1 16878.396,E2 16878.396} C_VEL
LIN {X 0,Y 358.404,Z 321.821,A -85,B 0,C 180,E1 16877.996,E2 16877.996} C_VEL
LIN {X 0,Y 373.606,Z 347.823,A -85,B 0,C 180,E1 16875.237,E2 16875.237} C_VEL
LIN {X 0,Y 383.238,Z 365.509,A -85,B 0,C 180,E1 16873.601,E2 16873.601} C_VEL
LIN {X 0,Y 372.019,Z 577.042,A -85,B 0,C 180,E1 16868.603,E2 16868.603} C_VEL
LIN {X 0,Y 370.171,Z 598.602,A -85,B 0,C 180,E1 16867.821,E2 16867.821} C_VEL
LIN {X 0,Y 367.915,Z 618.856,A -85,B 0,C 180,E1 16866.813,E2 16866.813} C_VEL
LIN {X 0,Y 365.208,Z 639.397,A -85,B 0,C 180,E1 16865.477,E2 16865.477} C_VEL
LIN {X 0,Y 362.281,Z 658.87,A -85,B 0,C 180,E1 16863.88,E2 16863.88} C_VEL
LIN {X 0,Y 359.223,Z 677.349,A -85,B 0,C 180,E1 16862.019,E2 16862.019} C_VEL
LIN {X 0,Y 356.067,Z 695.384,A -85,B 0,C 180,E1 16859.809,E2 16859.809} C_VEL
LIN {X 0,Y 353.131,Z 711.686,A -85,B 0,C 180,E1 16857.391,E2 16857.391} C_VEL
LIN {X 0,Y 350.53,Z 726.275,A -85,B 0,C 180,E1 16854.788,E2 16854.788} C_VEL
LIN {X 0,Y 348.314,Z 739.285,A -85,B 0,C 180,E1 16852,E2 16852} C_VEL
LIN {X 0,Y 346.642,Z 750.137,A -85,B 0,C 180,E1 16849.195,E2 16849.195} C_VEL
LIN {X 0,Y 345.37,Z 759.868,A -85,B 0,C 180,E1 16846.134,E2 16846.134} C_VEL
LIN {X 0,Y 344.543,Z 768.036,A -85,B 0,C 180,E1 16842.91,E2 16842.91} C_VEL
LIN {X 0,Y 344.17,Z 773.995,A -85,B 0,C 180,E1 16839.867,E2 16839.867} C_VEL
LIN {X 0,Y 344.051,Z 778.52,A -85,B 0,C 180,E1 16836.674,E2 16836.674} C_VEL
LIN {X 0,Y 344.057,Z 781.236,A -85,B 0,C 180,E1 16833.497,E2 16833.497} C_VEL
LIN {X 0,Y 344.083,Z 782.274,A -85,B 0,C 180,E1 16830.498,E2 16830.498} C_VEL
LIN {X 0,Y 344.063,Z 781.868,A -85,B 0,C 180,E1 16827.5,E2 16827.5} C_VEL
LIN {X 0,Y 344.03,Z 779.915,A -85,B 0,C 180,E1 16824.495,E2 16824.495} C_VEL
LIN {X 0,Y 344.093,Z 776.22,A -85,B 0,C 180,E1 16821.308,E2 16821.308} C_VEL
LIN {X 0,Y 344.378,Z 770.757,A -85,B 0,C 180,E1 16818.078,E2 16818.078} C_VEL
LIN {X 0,Y 345.064,Z 763.554,A -85,B 0,C 180,E1 16814.882,E2 16814.882} C_VEL
LIN {X 0,Y 346.199,Z 754.865,A -85,B 0,C 180,E1 16811.824,E2 16811.824} C_VEL
LIN {X 0,Y 347.906,Z 744.129,A -85,B 0,C 180,E1 16808.768,E2 16808.768} C_VEL
LIN {X 0,Y 350.105,Z 731.892,A -85,B 0,C 180,E1 16805.895,E2 16805.895} C_VEL
LIN {X 0,Y 352.759,Z 718.215,A -85,B 0,C 180,E1 16803.212,E2 16803.212} C_VEL
LIN {X 0,Y 355.919,Z 702.579,A -85,B 0,C 180,E1 16800.644,E2 16800.644} C_VEL
LIN {X 0,Y 359.23,Z 686.232,A -85,B 0,C 180,E1 16798.396,E2 16798.396} C_VEL
LIN {X 0,Y 362.896,Z 667.84,A -85,B 0,C 180,E1 16796.285,E2 16796.285} C_VEL
LIN {X 0,Y 366.559,Z 648.799,A -85,B 0,C 180,E1 16794.478,E2 16794.478} C_VEL
LIN {X 0,Y 370.291,Z 628.255,A -85,B 0,C 180,E1 16792.878,E2 16792.878} C_VEL
LIN {X 0,Y 373.881,Z 607.142,A -85,B 0,C 180,E1 16791.563,E2 16791.563} C_VEL
LIN {X 0,Y 377.388,Z 584.513,A -85,B 0,C 180,E1 16790.474,E2 16790.474} C_VEL
LIN {X 0,Y 380.743,Z 558.283,A -85,B 0,C 180,E1 16789.547,E2 16789.547} C_VEL
LIN {X 0,Y 387.733,Z 506.206,A -85,B 0,C 180,E1 16787.827,E2 16787.827} C_VEL
LIN {X 0,Y 396.994,Z 453.329,A -85,B 0,C 180,E1 16785.999,E2 16785.999} C_VEL
LIN {X 0,Y 409.103,Z 397.946,A -85,B 0,C 180,E1 16784.089,E2 16784.089} C_VEL
LIN {X 0,Y 412.398,Z 384.444,A -85,B 0,C 180,E1 16783.637,E2 16783.637} C_VEL
LIN {X 0,Y 412.031,Z 385.987,A -85,B 0,C 180,E1 16782.565,E2 16782.565} C_VEL
LIN {X 0,Y 411.881,Z 386.988,A -85,B 0,C 180,E1 16782.313,E2 16782.313} C_VEL
LIN {X 0,Y 410.876,Z 391.512,A -85,B 0,C 180,E1 16782.017,E2 16782.017} C_VEL
LIN {X 0,Y 395.678,Z 460.676,A -85,B 0,C 180,E1 16779.599,E2 16779.599} C_VEL
LIN {X 0,Y 384.652,Z 522.343,A -85,B 0,C 180,E1 16777.363,E2 16777.363} C_VEL
LIN {X 0,Y 377.025,Z 574.21,A -85,B 0,C 180,E1 16775.447,E2 16775.447} C_VEL
LIN {X 0,Y 373.634,Z 595.093,A -85,B 0,C 180,E1 16774.377,E2 16774.377} C_VEL
LIN {X 0,Y 369.925,Z 615.815,A -85,B 0,C 180,E1 16772.999,E2 16772.999} C_VEL
LIN {X 0,Y 366.124,Z 635.487,A -85,B 0,C 180,E1 16771.348,E2 16771.348} C_VEL
LIN {X 0,Y 362.315,Z 654.128,A -85,B 0,C 180,E1 16769.42,E2 16769.42} C_VEL
LIN {X 0,Y 358.85,Z 670.387,A -85,B 0,C 180,E1 16767.37,E2 16767.37} C_VEL
LIN {X 0,Y 355.516,Z 685.664,A -85,B 0,C 180,E1 16765.041,E2 16765.041} C_VEL
LIN {X 0,Y 352.515,Z 699.304,A -85,B 0,C 180,E1 16762.513,E2 16762.513} C_VEL
LIN {X 0,Y 349.988,Z 710.975,A -85,B 0,C 180,E1 16759.874,E2 16759.874} C_VEL
LIN {X 0,Y 347.892,Z 721.126,A -85,B 0,C 180,E1 16757.046,E2 16757.046} C_VEL
LIN {X 0,Y 346.356,Z 729.292,A -85,B 0,C 180,E1 16754.204,E2 16754.204} C_VEL
LIN {X 0,Y 345.258,Z 735.992,A -85,B 0,C 180,E1 16751.188,E2 16751.188} C_VEL
LIN {X 0,Y 344.6,Z 740.879,A -85,B 0,C 180,E1 16748.173,E2 16748.173} C_VEL
LIN {X 0,Y 344.253,Z 744.174,A -85,B 0,C 180,E1 16744.998,E2 16744.998} C_VEL
LIN {X 0,Y 344.12,Z 745.622,A -85,B 0,C 180,E1 16741.998,E2 16741.998} C_VEL
LIN {X 0,Y 344.09,Z 745.431,A -85,B 0,C 180,E1 16739,E2 16739} C_VEL
LIN {X 0,Y 344.109,Z 743.619,A -85,B 0,C 180,E1 16736.001,E2 16736.001} C_VEL
LIN {X 0,Y 344.264,Z 740.153,A -85,B 0,C 180,E1 16732.993,E2 16732.993} C_VEL
LIN {X 0,Y 344.659,Z 734.945,A -85,B 0,C 180,E1 16729.975,E2 16729.975} C_VEL
LIN {X 0,Y 345.34,Z 728.301,A -85,B 0,C 180,E1 16727.118,E2 16727.118} C_VEL
LIN {X 0,Y 346.434,Z 719.818,A -85,B 0,C 180,E1 16724.258,E2 16724.258} C_VEL
LIN {X 0,Y 347.954,Z 709.604,A -85,B 0,C 180,E1 16721.493,E2 16721.493} C_VEL
LIN {X 0,Y 349.858,Z 697.859,A -85,B 0,C 180,E1 16718.893,E2 16718.893} C_VEL
LIN {X 0,Y 351.998,Z 685.158,A -85,B 0,C 180,E1 16716.564,E2 16716.564} C_VEL
LIN {X 0,Y 354.456,Z 670.589,A -85,B 0,C 180,E1 16714.341,E2 16714.341} C_VEL
LIN {X 0,Y 357.092,Z 654.42,A -85,B 0,C 180,E1 16712.302,E2 16712.302} C_VEL
LIN {X 0,Y 359.73,Z 637.257,A -85,B 0,C 180,E1 16710.529,E2 16710.529} C_VEL
LIN {X 0,Y 362.248,Z 619.175,A -85,B 0,C 180,E1 16709.017,E2 16709.017} C_VEL
LIN {X 0,Y 364.563,Z 599.974,A -85,B 0,C 180,E1 16707.752,E2 16707.752} C_VEL
LIN {X 0,Y 366.567,Z 579.862,A -85,B 0,C 180,E1 16706.752,E2 16706.752} C_VEL
LIN {X 0,Y 368.1,Z 559.726,A -85,B 0,C 180,E1 16706.045,E2 16706.045} C_VEL
LIN {X 0,Y 377.641,Z 380.802,A -85,B 0,C 180,E1 16701.636,E2 16701.636} C_VEL
LIN {X 0,Y 374.683,Z 359.244,A -85,B 0,C 180,E1 16700.645,E2 16700.645} C_VEL
LIN {X 0,Y 363.805,Z 338.545,A -85,B 0,C 180,E1 16698.677,E2 16698.677} C_VEL
LIN {X 0,Y 356.684,Z 319.845,A -85,B 0,C 180,E1 16695.172,E2 16695.172} C_VEL
LIN {X 0,Y 350.22,Z 304.007,A -85,B 0,C 180,E1 16691.919,E2 16691.919} C_VEL
LIN {X 0,Y 345.957,Z 293.592,A -85,B 0,C 180,E1 16689.58,E2 16689.58} C_VEL
LIN {X 0,Y 345.924,Z 293.396,A -85,B 0,C 180,E1 16685.317,E2 16685.317} C_VEL
LIN {X 0,Y 345.917,Z 293.39,A -85,B 0,C 180,E1 16681.159,E2 16681.159} C_VEL
LIN {X 0,Y 345.907,Z 293.399,A -85,B 0,C 180,E1 16676.99,E2 16676.99} C_VEL
LIN {X 0,Y 345.959,Z 293.599,A -85,B 0,C 180,E1 16674.14,E2 16674.14} C_VEL
LIN {X 0,Y 346.386,Z 295.233,A -85,B 0,C 180,E1 16673.788,E2 16673.788} C_VEL
LIN {X 0,Y 351.277,Z 305.801,A -85,B 0,C 180,E1 16671.886,E2 16671.886} C_VEL
LIN {X 0,Y 358.505,Z 323.211,A -85,B 0,C 180,E1 16669.008,E2 16669.008} C_VEL
LIN {X 0,Y 364.738,Z 340.658,A -85,B 0,C 180,E1 16666.368,E2 16666.368} C_VEL
LIN {X 0,Y 367.575,Z 349.984,A -85,B 0,C 180,E1 16665.057,E2 16665.057} C_VEL
LIN {X 0,Y 364.449,Z 392.246,A -85,B 0,C 180,E1 16660.914,E2 16660.914} C_VEL
LIN {X 0,Y 361.378,Z 433.081,A -85,B 0,C 180,E1 16656.914,E2 16656.914} C_VEL
LIN {X 0,Y 358.449,Z 474.145,A -85,B 0,C 180,E1 16652.88,E2 16652.88} C_VEL
LIN {X 0,Y 358.077,Z 481.347,A -85,B 0,C 180,E1 16652.226,E2 16652.226} C_VEL
LIN {X 0,Y 359.22,Z 491.389,A -85,B 0,C 180,E1 16651.911,E2 16651.911} C_VEL
LIN {X 0,Y 359.056,Z 497.957,A -85,B 0,C 180,E1 16651.777,E2 16651.777} C_VEL
LIN {X 0,Y 356.653,Z 507.714,A -85,B 0,C 180,E1 16651.745,E2 16651.745} C_VEL
LIN {X 0,Y 352.824,Z 520.75,A -85,B 0,C 180,E1 16651.748,E2 16651.748} C_VEL
LIN {X 0,Y 352.141,Z 526.316,A -85,B 0,C 180,E1 16651.675,E2 16651.675} C_VEL
LIN {X 0,Y 349.599,Z 625.09,A -85,B 0,C 180,E1 16649.592,E2 16649.592} C_VEL
LIN {X 0,Y 348.789,Z 641.248,A -85,B 0,C 180,E1 16648.95,E2 16648.95} C_VEL
LIN {X 0,Y 347.603,Z 656.897,A -85,B 0,C 180,E1 16648.024,E2 16648.024} C_VEL
LIN {X 0,Y 346.15,Z 671.38,A -85,B 0,C 180,E1 16646.856,E2 16646.856} C_VEL
LIN {X 0,Y 344.413,Z 685.801,A -85,B 0,C 180,E1 16645.339,E2 16645.339} C_VEL
LIN {X 0,Y 342.68,Z 698.496,A -85,B 0,C 180,E1 16643.636,E2 16643.636} C_VEL
LIN {X 0,Y 340.907,Z 710.688,A -85,B 0,C 180,E1 16641.569,E2 16641.569} C_VEL
LIN {X 0,Y 339.442,Z 720.467,A -85,B 0,C 180,E1 16639.479,E2 16639.479} C_VEL
LIN {X 0,Y 338.122,Z 729.538,A -85,B 0,C 180,E1 16637.015,E2 16637.015} C_VEL
LIN {X 0,Y 337.19,Z 736.557,A -85,B 0,C 180,E1 16634.52,E2 16634.52} C_VEL
LIN {X 0,Y 336.572,Z 742.076,A -85,B 0,C 180,E1 16631.827,E2 16631.827} C_VEL
LIN {X 0,Y 336.275,Z 745.59,A -85,B 0,C 180,E1 16629.281,E2 16629.281} C_VEL
LIN {X 0,Y 336.147,Z 747.599,A -85,B 0,C 180,E1 16626.513,E2 16626.513} C_VEL
LIN {X 0,Y 336.151,Z 747.893,A -85,B 0,C 180,E1 16623.695,E2 16623.695} C_VEL
LIN {X 0,Y 336.277,Z 746.368,A -85,B 0,C 180,E1 16620.947,E2 16620.947} C_VEL
LIN {X 0,Y 336.636,Z 742.95,A -85,B 0,C 180,E1 16618.086,E2 16618.086} C_VEL
LIN {X 0,Y 337.256,Z 738.038,A -85,B 0,C 180,E1 16615.507,E2 16615.507} C_VEL
LIN {X 0,Y 338.268,Z 731.244,A -85,B 0,C 180,E1 16612.919,E2 16612.919} C_VEL
LIN {X 0,Y 339.608,Z 722.889,A -85,B 0,C 180,E1 16610.513,E2 16610.513} C_VEL
LIN {X 0,Y 341.323,Z 712.507,A -85,B 0,C 180,E1 16608.184,E2 16608.184} C_VEL
LIN {X 0,Y 343.099,Z 701.367,A -85,B 0,C 180,E1 16606.216,E2 16606.216} C_VEL
LIN {X 0,Y 345.017,Z 688.531,A -85,B 0,C 180,E1 16604.411,E2 16604.411} C_VEL
LIN {X 0,Y 346.793,Z 675.042,A -85,B 0,C 180,E1 16602.922,E2 16602.922} C_VEL
LIN {X 0,Y 348.486,Z 659.851,A -85,B 0,C 180,E1 16601.632,E2 16601.632} C_VEL
LIN {X 0,Y 349.777,Z 644.4,A -85,B 0,C 180,E1 16600.669,E2 16600.669} C_VEL
LIN {X 0,Y 350.718,Z 627.649,A -85,B 0,C 180,E1 16599.959,E2 16599.959} C_VEL
LIN {X 0,Y 351.621,Z 594.862,A -85,B 0,C 180,E1 16599.214,E2 16599.214} C_VEL
LIN {X 0,Y 354.151,Z 499.226,A -85,B 0,C 180,E1 16597.199,E2 16597.199} C_VEL
LIN {X 0,Y 352.226,Z 481.476,A -85,B 0,C 180,E1 16596.553,E2 16596.553} C_VEL
LIN {X 0,Y 355.443,Z 439.199,A -85,B 0,C 180,E1 16592.404,E2 16592.404} C_VEL
LIN {X 0,Y 358.764,Z 397.06,A -85,B 0,C 180,E1 16588.281,E2 16588.281} C_VEL
LIN {X 0,Y 361.791,Z 356.157,A -85,B 0,C 180,E1 16584.318,E2 16584.318} C_VEL
LIN {X 0,Y 361.858,Z 351.927,A -85,B 0,C 180,E1 16583.879,E2 16583.879} C_VEL
LIN {X 0,Y 356.589,Z 335.585,A -85,B 0,C 180,E1 16581.378,E2 16581.378} C_VEL
LIN {X 0,Y 350.621,Z 320.641,A -85,B 0,C 180,E1 16578.799,E2 16578.799} C_VEL
LIN {X 0,Y 344.779,Z 307.854,A -85,B 0,C 180,E1 16576.338,E2 16576.338} C_VEL
LIN {X 0,Y 339.802,Z 298.575,A -85,B 0,C 180,E1 16574.311,E2 16574.311} C_VEL
LIN {X 0,Y 338.114,Z 295.101,A -85,B 0,C 180,E1 16573.511,E2 16573.511} C_VEL
LIN {X 0,Y 337.989,Z 294.413,A -85,B 0,C 180,E1 16573.167,E2 16573.167} C_VEL
LIN {X 0,Y 337.971,Z 294.384,A -85,B 0,C 180,E1 16568.85,E2 16568.85} C_VEL
LIN {X 0,Y 337.964,Z 294.384,A -85,B 0,C 180,E1 16564.582,E2 16564.582} C_VEL
LIN {X 0,Y 337.962,Z 294.388,A -85,B 0,C 180,E1 16560.17,E2 16560.17} C_VEL
LIN {X 0,Y 337.964,Z 294.38,A -85,B 0,C 180,E1 16555.929,E2 16555.929} C_VEL
LIN {X 0,Y 337.974,Z 294.388,A -85,B 0,C 180,E1 16551.666,E2 16551.666} C_VEL
LIN {X 0,Y 337.985,Z 294.377,A -85,B 0,C 180,E1 16547.355,E2 16547.355} C_VEL
LIN {X 0,Y 337.991,Z 294.382,A -85,B 0,C 180,E1 16543.148,E2 16543.148} C_VEL
LIN {X 0,Y 337.991,Z 294.379,A -85,B 0,C 180,E1 16538.845,E2 16538.845} C_VEL
LIN {X 0,Y 337.98,Z 294.382,A -85,B 0,C 180,E1 16534.599,E2 16534.599} C_VEL
LIN {X 0,Y 337.975,Z 294.381,A -85,B 0,C 180,E1 16530.394,E2 16530.394} C_VEL
LIN {X 0,Y 337.972,Z 294.383,A -85,B 0,C 180,E1 16526.209,E2 16526.209} C_VEL
LIN {X 0,Y 338.024,Z 294.627,A -85,B 0,C 180,E1 16524.775,E2 16524.775} C_VEL
LIN {X 0,Y 340.974,Z 301.625,A -85,B 0,C 180,E1 16523.177,E2 16523.177} C_VEL
LIN {X 0,Y 348.1,Z 317.658,A -85,B 0,C 180,E1 16519.818,E2 16519.818} C_VEL
LIN {X 0,Y 349.811,Z 321.321,A -85,B 0,C 180,E1 16519.169,E2 16519.169} C_VEL
LIN {X 0,Y 364.926,Z 347.052,A -85,B 0,C 180,E1 16516.307,E2 16516.307} C_VEL
LIN {X 0,Y 376.628,Z 368.263,A -85,B 0,C 180,E1 16514.252,E2 16514.252} C_VEL
LIN {X 0,Y 364.998,Z 577.035,A -85,B 0,C 180,E1 16509.2,E2 16509.2} C_VEL
LIN {X 0,Y 363.082,Z 598.522,A -85,B 0,C 180,E1 16508.404,E2 16508.404} C_VEL
LIN {X 0,Y 360.736,Z 618.858,A -85,B 0,C 180,E1 16507.371,E2 16507.371} C_VEL
LIN {X 0,Y 357.939,Z 639.326,A -85,B 0,C 180,E1 16506.013,E2 16506.013} C_VEL
LIN {X 0,Y 354.853,Z 659.156,A -85,B 0,C 180,E1 16504.354,E2 16504.354} C_VEL
LIN {X 0,Y 351.544,Z 678.422,A -85,B 0,C 180,E1 16502.358,E2 16502.358} C_VEL
LIN {X 0,Y 348.361,Z 695.927,A -85,B 0,C 180,E1 16500.149,E2 16500.149} C_VEL
LIN {X 0,Y 345.347,Z 712.086,A -85,B 0,C 180,E1 16497.687,E2 16497.687} C_VEL
LIN {X 0,Y 342.668,Z 726.607,A -85,B 0,C 180,E1 16495.027,E2 16495.027} C_VEL
LIN {X 0,Y 340.328,Z 739.902,A -85,B 0,C 180,E1 16492.087,E2 16492.087} C_VEL
LIN {X 0,Y 338.498,Z 751.508,A -85,B 0,C 180,E1 16488.958,E2 16488.958} C_VEL
LIN {X 0,Y 337.256,Z 760.909,A -85,B 0,C 180,E1 16485.826,E2 16485.826} C_VEL
LIN {X 0,Y 336.506,Z 768.386,A -85,B 0,C 180,E1 16482.7,E2 16482.7} C_VEL
LIN {X 0,Y 336.14,Z 774.404,A -85,B 0,C 180,E1 16479.414,E2 16479.414} C_VEL
LIN {X 0,Y 336.06,Z 778.451,A -85,B 0,C 180,E1 16476.318,E2 16476.318} C_VEL
LIN {X 0,Y 336.071,Z 780.929,A -85,B 0,C 180,E1 16473.239,E2 16473.239} C_VEL
LIN {X 0,Y 336.104,Z 781.831,A -85,B 0,C 180,E1 16470.169,E2 16470.169} C_VEL
LIN {X 0,Y 336.064,Z 781.192,A -85,B 0,C 180,E1 16466.928,E2 16466.928} C_VEL
LIN {X 0,Y 336.04,Z 779.085,A -85,B 0,C 180,E1 16463.849,E2 16463.849} C_VEL
LIN {X 0,Y 336.123,Z 775.131,A -85,B 0,C 180,E1 16460.582,E2 16460.582} C_VEL
LIN {X 0,Y 336.501,Z 769.44,A -85,B 0,C 180,E1 16457.296,E2 16457.296} C_VEL
LIN {X 0,Y 337.345,Z 761.904,A -85,B 0,C 180,E1 16453.998,E2 16453.998} C_VEL
LIN {X 0,Y 338.672,Z 752.894,A -85,B 0,C 180,E1 16450.861,E2 16450.861} C_VEL
LIN {X 0,Y 340.502,Z 742.618,A -85,B 0,C 180,E1 16447.921,E2 16447.921} C_VEL
LIN {X 0,Y 342.955,Z 730.241,A -85,B 0,C 180,E1 16444.991,E2 16444.991} C_VEL
LIN {X 0,Y 346.083,Z 715.492,A -85,B 0,C 180,E1 16442.092,E2 16442.092} C_VEL
LIN {X 0,Y 349.707,Z 698.984,A -85,B 0,C 180,E1 16439.406,E2 16439.406} C_VEL
LIN {X 0,Y 353.621,Z 681.141,A -85,B 0,C 180,E1 16437,E2 16437} C_VEL
LIN {X 0,Y 357.655,Z 662.442,A -85,B 0,C 180,E1 16434.912,E2 16434.912} C_VEL
LIN {X 0,Y 361.835,Z 642.249,A -85,B 0,C 180,E1 16433.056,E2 16433.056} C_VEL
LIN {X 0,Y 366.004,Z 621.018,A -85,B 0,C 180,E1 16431.473,E2 16431.473} C_VEL
LIN {X 0,Y 370.038,Z 599.043,A -85,B 0,C 180,E1 16430.178,E2 16430.178} C_VEL
LIN {X 0,Y 373.917,Z 575.802,A -85,B 0,C 180,E1 16429.138,E2 16429.138} C_VEL
LIN {X 0,Y 383.569,Z 511.855,A -85,B 0,C 180,E1 16426.923,E2 16426.923} C_VEL
LIN {X 0,Y 393.837,Z 459.479,A -85,B 0,C 180,E1 16425.068,E2 16425.068} C_VEL
LIN {X 0,Y 407.154,Z 404.303,A -85,B 0,C 180,E1 16423.154,E2 16423.154} C_VEL
LIN {X 0,Y 408.739,Z 398.253,A -85,B 0,C 180,E1 16422.934,E2 16422.934} C_VEL
LIN {X 0,Y 392.321,Z 466.817,A -85,B 0,C 180,E1 16420.52,E2 16420.52} C_VEL
LIN {X 0,Y 380.562,Z 526.134,A -85,B 0,C 180,E1 16418.319,E2 16418.319} C_VEL
LIN {X 0,Y 372.421,Z 575.002,A -85,B 0,C 180,E1 16416.441,E2 16416.441} C_VEL
LIN {X 0,Y 368.501,Z 596.344,A -85,B 0,C 180,E1 16415.305,E2 16415.305} C_VEL
LIN {X 0,Y 364.502,Z 616.293,A -85,B 0,C 180,E1 16413.932,E2 16413.932} C_VEL
LIN {X 0,Y 360.215,Z 636.313,A -85,B 0,C 180,E1 16412.204,E2 16412.204} C_VEL
LIN {X 0,Y 355.961,Z 655.265,A -85,B 0,C 180,E1 16410.184,E2 16410.184} C_VEL
LIN {X 0,Y 352.113,Z 671.811,A -85,B 0,C 180,E1 16408.031,E2 16408.031} C_VEL
LIN {X 0,Y 348.545,Z 686.8,A -85,B 0,C 180,E1 16405.668,E2 16405.668} C_VEL
LIN {X 0,Y 345.219,Z 700.605,A -85,B 0,C 180,E1 16403.016,E2 16403.016} C_VEL
LIN {X 0,Y 342.512,Z 712.08,A -85,B 0,C 180,E1 16400.327,E2 16400.327} C_VEL
LIN {X 0,Y 340.26,Z 722.087,A -85,B 0,C 180,E1 16397.441,E2 16397.441} C_VEL
LIN {X 0,Y 338.593,Z 730.136,A -85,B 0,C 180,E1 16394.536,E2 16394.536} C_VEL
LIN {X 0,Y 337.395,Z 736.734,A -85,B 0,C 180,E1 16391.452,E2 16391.452} C_VEL
LIN {X 0,Y 336.673,Z 741.533,A -85,B 0,C 180,E1 16388.367,E2 16388.367} C_VEL
LIN {X 0,Y 336.303,Z 744.635,A -85,B 0,C 180,E1 16385.288,E2 16385.288} C_VEL
LIN {X 0,Y 336.142,Z 746.084,A -85,B 0,C 180,E1 16382.215,E2 16382.215} C_VEL
LIN {X 0,Y 336.101,Z 745.899,A -85,B 0,C 180,E1 16379.147,E2 16379.147} C_VEL
LIN {X 0,Y 336.118,Z 744.091,A -85,B 0,C 180,E1 16376.076,E2 16376.076} C_VEL
LIN {X 0,Y 336.274,Z 740.622,A -85,B 0,C 180,E1 16372.997,E2 16372.997} C_VEL
LIN {X 0,Y 336.682,Z 735.404,A -85,B 0,C 180,E1 16369.908,E2 16369.908} C_VEL
LIN {X 0,Y 337.391,Z 728.745,A -85,B 0,C 180,E1 16366.983,E2 16366.983} C_VEL
LIN {X 0,Y 338.53,Z 720.238,A -85,B 0,C 180,E1 16364.056,E2 16364.056} C_VEL
LIN {X 0,Y 340.144,Z 709.81,A -85,B 0,C 180,E1 16361.181,E2 16361.181} C_VEL
LIN {X 0,Y 342.094,Z 698.219,A -85,B 0,C 180,E1 16358.57,E2 16358.57} C_VEL
LIN {X 0,Y 344.355,Z 685.278,A -85,B 0,C 180,E1 16356.155,E2 16356.155} C_VEL
LIN {X 0,Y 346.975,Z 670.305,A -85,B 0,C 180,E1 16353.838,E2 16353.838} C_VEL
LIN {X 0,Y 349.725,Z 653.999,A -85,B 0,C 180,E1 16351.759,E2 16351.759} C_VEL
LIN {X 0,Y 352.47,Z 636.673,A -85,B 0,C 180,E1 16349.954,E2 16349.954} C_VEL
LIN {X 0,Y 355.169,Z 617.678,A -85,B 0,C 180,E1 16348.367,E2 16348.367} C_VEL
LIN {X 0,Y 357.551,Z 598.311,A -85,B 0,C 180,E1 16347.097,E2 16347.097} C_VEL
LIN {X 0,Y 359.582,Z 578.331,A -85,B 0,C 180,E1 16346.109,E2 16346.109} C_VEL
LIN {X 0,Y 361.197,Z 557.274,A -85,B 0,C 180,E1 16345.383,E2 16345.383} C_VEL
LIN {X 0,Y 371.023,Z 381.928,A -85,B 0,C 180,E1 16340.955,E2 16340.955} C_VEL
LIN {X 0,Y 368.342,Z 362.58,A -85,B 0,C 180,E1 16340.043,E2 16340.043} C_VEL
LIN {X 0,Y 355.537,Z 338.327,A -85,B 0,C 180,E1 16337.641,E2 16337.641} C_VEL
LIN {X 0,Y 348.076,Z 318.918,A -85,B 0,C 180,E1 16333.861,E2 16333.861} C_VEL
LIN {X 0,Y 340.999,Z 301.781,A -85,B 0,C 180,E1 16330.173,E2 16330.173} C_VEL
LIN {X 0,Y 338.021,Z 294.573,A -85,B 0,C 180,E1 16328.462,E2 16328.462} C_VEL
LIN {X 0,Y 337.992,Z 294.383,A -85,B 0,C 180,E1 16324.074,E2 16324.074} C_VEL
LIN {X 0,Y 337.995,Z 294.356,A -85,B 0,C 180,E1 16319.802,E2 16319.802} C_VEL
LIN {X 0,Y 337.978,Z 294.364,A -85,B 0,C 180,E1 16315.536,E2 16315.536} C_VEL
LIN {X 0,Y 338.035,Z 294.816,A -85,B 0,C 180,E1 16315.118,E2 16315.118} C_VEL
LIN {X 0,Y 339.459,Z 298.103,A -85,B 0,C 180,E1 16314.473,E2 16314.473} C_VEL
LIN {X 0,Y 346.624,Z 313.982,A -85,B 0,C 180,E1 16311.589,E2 16311.589} C_VEL
LIN {X 0,Y 353.778,Z 331.98,A -85,B 0,C 180,E1 16308.626,E2 16308.626} C_VEL
LIN {X 0,Y 359.704,Z 349.633,A -85,B 0,C 180,E1 16305.975,E2 16305.975} C_VEL
LIN {X 0,Y 360.6,Z 352.898,A -85,B 0,C 180,E1 16305.521,E2 16305.521} C_VEL
LIN {X 0,Y 357.417,Z 393.918,A -85,B 0,C 180,E1 16301.458,E2 16301.458} C_VEL
LIN {X 0,Y 354.17,Z 435.046,A -85,B 0,C 180,E1 16297.382,E2 16297.382} C_VEL
LIN {X 0,Y 351.013,Z 477.267,A -85,B 0,C 180,E1 16293.186,E2 16293.186} C_VEL
LIN {X 0,Y 350.845,Z 481.781,A -85,B 0,C 180,E1 16292.799,E2 16292.799} C_VEL
LIN {X 0,Y 352.802,Z 501.673,A -85,B 0,C 180,E1 16292.184,E2 16292.184} C_VEL
LIN {X 0,Y 352.141,Z 526.316,A -85,B 0,C 180,E1 16291.675,E2 16291.675} C_VEL
LIN {X 0,Y 351.015,Z 533.985,A -85,B 0,C 180,E1 16291.589,E2 16291.589} C_VEL
LIN {X 0,Y 344.857,Z 554.319,A -85,B 0,C 180,E1 16291.607,E2 16291.607} C_VEL
LIN {X 0,Y 344.007,Z 560.903,A -85,B 0,C 180,E1 16291.522,E2 16291.522} C_VEL
LIN {X 0,Y 342.252,Z 625.857,A -85,B 0,C 180,E1 16290.106,E2 16290.106} C_VEL
LIN {X 0,Y 341.382,Z 642.145,A -85,B 0,C 180,E1 16289.436,E2 16289.436} C_VEL
LIN {X 0,Y 340.083,Z 658.406,A -85,B 0,C 180,E1 16288.44,E2 16288.44} C_VEL
LIN {X 0,Y 338.416,Z 673.874,A -85,B 0,C 180,E1 16287.123,E2 16287.123} C_VEL
LIN {X 0,Y 336.627,Z 687.872,A -85,B 0,C 180,E1 16285.573,E2 16285.573} C_VEL
LIN {X 0,Y 334.761,Z 700.769,A -85,B 0,C 180,E1 16283.743,E2 16283.743} C_VEL
LIN {X 0,Y 333.014,Z 712.162,A -85,B 0,C 180,E1 16281.716,E2 16281.716} C_VEL
LIN {X 0,Y 331.394,Z 722.426,A -85,B 0,C 180,E1 16279.397,E2 16279.397} C_VEL
LIN {X 0,Y 330.153,Z 730.631,A -85,B 0,C 180,E1 16277.052,E2 16277.052} C_VEL
LIN {X 0,Y 329.155,Z 737.778,A -85,B 0,C 180,E1 16274.355,E2 16274.355} C_VEL
LIN {X 0,Y 328.566,Z 742.901,A -85,B 0,C 180,E1 16271.706,E2 16271.706} C_VEL
LIN {X 0,Y 328.257,Z 746.362,A -85,B 0,C 180,E1 16268.938,E2 16268.938} C_VEL
LIN {X 0,Y 328.15,Z 748.169,A -85,B 0,C 180,E1 16266.078,E2 16266.078} C_VEL
LIN {X 0,Y 328.166,Z 748.212,A -85,B 0,C 180,E1 16263.395,E2 16263.395} C_VEL
LIN {X 0,Y 328.335,Z 746.434,A -85,B 0,C 180,E1 16260.443,E2 16260.443} C_VEL
LIN {X 0,Y 328.737,Z 742.939,A -85,B 0,C 180,E1 16257.638,E2 16257.638} C_VEL
LIN {X 0,Y 329.516,Z 737.416,A -85,B 0,C 180,E1 16254.797,E2 16254.797} C_VEL
LIN {X 0,Y 330.577,Z 730.877,A -85,B 0,C 180,E1 16252.344,E2 16252.344} C_VEL
LIN {X 0,Y 332.118,Z 721.88,A -85,B 0,C 180,E1 16249.78,E2 16249.78} C_VEL
LIN {X 0,Y 333.86,Z 711.932,A -85,B 0,C 180,E1 16247.562,E2 16247.562} C_VEL
LIN {X 0,Y 335.853,Z 699.998,A -85,B 0,C 180,E1 16245.468,E2 16245.468} C_VEL
LIN {X 0,Y 337.763,Z 687.766,A -85,B 0,C 180,E1 16243.759,E2 16243.759} C_VEL
LIN {X 0,Y 339.691,Z 673.523,A -85,B 0,C 180,E1 16242.203,E2 16242.203} C_VEL
LIN {X 0,Y 341.315,Z 659.407,A -85,B 0,C 180,E1 16241.011,E2 16241.011} C_VEL
LIN {X 0,Y 342.676,Z 643.422,A -85,B 0,C 180,E1 16240.024,E2 16240.024} C_VEL
LIN {X 0,Y 343.599,Z 627.214,A -85,B 0,C 180,E1 16239.344,E2 16239.344} C_VEL
LIN {X 0,Y 345.216,Z 570.976,A -85,B 0,C 180,E1 16238.092,E2 16238.092} C_VEL
LIN {X 0,Y 347.175,Z 499.948,A -85,B 0,C 180,E1 16236.559,E2 16236.559} C_VEL
LIN {X 0,Y 345.23,Z 482.09,A -85,B 0,C 180,E1 16235.898,E2 16235.898} C_VEL
LIN {X 0,Y 348.72,Z 438.304,A -85,B 0,C 180,E1 16231.553,E2 16231.553} C_VEL
LIN {X 0,Y 351.971,Z 398.894,A -85,B 0,C 180,E1 16227.667,E2 16227.667} C_VEL
LIN {X 0,Y 355.002,Z 360.835,A -85,B 0,C 180,E1 16223.928,E2 16223.928} C_VEL
LIN {X 0,Y 355.314,Z 355.414,A -85,B 0,C 180,E1 16223.377,E2 16223.377} C_VEL
LIN {X 0,Y 350.277,Z 339.623,A -85,B 0,C 180,E1 16220.905,E2 16220.905} C_VEL
LIN {X 0,Y 344.773,Z 325.615,A -85,B 0,C 180,E1 16218.428,E2 16218.428} C_VEL
LIN {X 0,Y 338.807,Z 312.634,A -85,B 0,C 180,E1 16215.842,E2 16215.842} C_VEL
LIN {X 0,Y 334.604,Z 304.41,A -85,B 0,C 180,E1 16214.008,E2 16214.008} C_VEL
LIN {X 0,Y 332,Z 299.711,A -85,B 0,C 180,E1 16212.878,E2 16212.878} C_VEL
LIN {X 0,Y 330.195,Z 296.3,A -85,B 0,C 180,E1 16212.041,E2 16212.041} C_VEL
LIN {X 0,Y 330.046,Z 295.41,A -85,B 0,C 180,E1 16211.637,E2 16211.637} C_VEL
LIN {X 0,Y 330.062,Z 295.372,A -85,B 0,C 180,E1 16207.31,E2 16207.31} C_VEL
LIN {X 0,Y 330.038,Z 295.376,A -85,B 0,C 180,E1 16202.953,E2 16202.953} C_VEL
LIN {X 0,Y 330.027,Z 295.369,A -85,B 0,C 180,E1 16198.612,E2 16198.612} C_VEL
LIN {X 0,Y 330.023,Z 295.376,A -85,B 0,C 180,E1 16194.263,E2 16194.263} C_VEL
LIN {X 0,Y 330.026,Z 295.368,A -85,B 0,C 180,E1 16189.88,E2 16189.88} C_VEL
LIN {X 0,Y 330.038,Z 295.376,A -85,B 0,C 180,E1 16185.617,E2 16185.617} C_VEL
LIN {X 0,Y 330.048,Z 295.365,A -85,B 0,C 180,E1 16181.27,E2 16181.27} C_VEL
LIN {X 0,Y 330.059,Z 295.37,A -85,B 0,C 180,E1 16176.997,E2 16176.997} C_VEL
LIN {X 0,Y 330.042,Z 295.369,A -85,B 0,C 180,E1 16172.573,E2 16172.573} C_VEL
LIN {X 0,Y 330.036,Z 295.371,A -85,B 0,C 180,E1 16168.349,E2 16168.349} C_VEL
LIN {X 0,Y 330.069,Z 295.642,A -85,B 0,C 180,E1 16165.974,E2 16165.974} C_VEL
LIN {X 0,Y 331.671,Z 299.336,A -85,B 0,C 180,E1 16165.057,E2 16165.057} C_VEL
LIN {X 0,Y 339.158,Z 316.344,A -85,B 0,C 180,E1 16161.319,E2 16161.319} C_VEL
LIN {X 0,Y 341.505,Z 321.378,A -85,B 0,C 180,E1 16160.338,E2 16160.338} C_VEL
LIN {X 0,Y 357.451,Z 348.34,A -85,B 0,C 180,E1 16157.206,E2 16157.206} C_VEL
LIN {X 0,Y 370.048,Z 371.248,A -85,B 0,C 180,E1 16154.919,E2 16154.919} C_VEL
LIN {X 0,Y 357.996,Z 576.955,A -85,B 0,C 180,E1 16149.815,E2 16149.815} C_VEL
LIN {X 0,Y 355.992,Z 598.538,A -85,B 0,C 180,E1 16148.997,E2 16148.997} C_VEL
LIN {X 0,Y 353.569,Z 618.824,A -85,B 0,C 180,E1 16147.944,E2 16147.944} C_VEL
LIN {X 0,Y 350.696,Z 639.126,A -85,B 0,C 180,E1 16146.572,E2 16146.572} C_VEL
LIN {X 0,Y 347.572,Z 658.567,A -85,B 0,C 180,E1 16144.919,E2 16144.919} C_VEL
LIN {X 0,Y 344.166,Z 677.781,A -85,B 0,C 180,E1 16142.904,E2 16142.904} C_VEL
LIN {X 0,Y 340.909,Z 695.134,A -85,B 0,C 180,E1 16140.683,E2 16140.683} C_VEL
LIN {X 0,Y 337.768,Z 711.391,A -85,B 0,C 180,E1 16138.171,E2 16138.171} C_VEL
LIN {X 0,Y 334.968,Z 725.97,A -85,B 0,C 180,E1 16135.454,E2 16135.454} C_VEL
LIN {X 0,Y 332.525,Z 739.34,A -85,B 0,C 180,E1 16132.447,E2 16132.447} C_VEL
LIN {X 0,Y 330.674,Z 750.572,A -85,B 0,C 180,E1 16129.372,E2 16129.372} C_VEL
LIN {X 0,Y 329.371,Z 759.964,A -85,B 0,C 180,E1 16126.215,E2 16126.215} C_VEL
LIN {X 0,Y 328.56,Z 767.582,A -85,B 0,C 180,E1 16123.012,E2 16123.012} C_VEL
LIN {X 0,Y 328.163,Z 773.719,A -85,B 0,C 180,E1 16119.645,E2 16119.645} C_VEL
LIN {X 0,Y 328.074,Z 777.864,A -85,B 0,C 180,E1 16116.473,E2 16116.473} C_VEL
LIN {X 0,Y 328.085,Z 780.383,A -85,B 0,C 180,E1 16113.318,E2 16113.318} C_VEL
LIN {X 0,Y 328.118,Z 781.355,A -85,B 0,C 180,E1 16110.173,E2 16110.173} C_VEL
LIN {X 0,Y 328.075,Z 780.859,A -85,B 0,C 180,E1 16107.028,E2 16107.028} C_VEL
LIN {X 0,Y 328.045,Z 778.829,A -85,B 0,C 180,E1 16103.874,E2 16103.874} C_VEL
LIN {X 0,Y 328.116,Z 775.251,A -85,B 0,C 180,E1 16100.704,E2 16100.704} C_VEL
LIN {X 0,Y 328.493,Z 769.816,A -85,B 0,C 180,E1 16097.339,E2 16097.339} C_VEL
LIN {X 0,Y 329.298,Z 763.002,A -85,B 0,C 180,E1 16094.139,E2 16094.139} C_VEL
LIN {X 0,Y 330.734,Z 753.863,A -85,B 0,C 180,E1 16090.758,E2 16090.758} C_VEL
LIN {X 0,Y 332.904,Z 742.52,A -85,B 0,C 180,E1 16087.389,E2 16087.389} C_VEL
LIN {X 0,Y 335.725,Z 729.474,A -85,B 0,C 180,E1 16084.225,E2 16084.225} C_VEL
LIN {X 0,Y 339.122,Z 714.749,A -85,B 0,C 180,E1 16081.275,E2 16081.275} C_VEL
LIN {X 0,Y 343.041,Z 698.333,A -85,B 0,C 180,E1 16078.55,E2 16078.55} C_VEL
LIN {X 0,Y 347.215,Z 680.841,A -85,B 0,C 180,E1 16076.135,E2 16076.135} C_VEL
LIN {X 0,Y 351.726,Z 661.714,A -85,B 0,C 180,E1 16073.952,E2 16073.952} C_VEL
LIN {X 0,Y 356.386,Z 641.227,A -85,B 0,C 180,E1 16072.032,E2 16072.032} C_VEL
LIN {X 0,Y 360.995,Z 620.134,A -85,B 0,C 180,E1 16070.427,E2 16070.427} C_VEL
LIN {X 0,Y 365.603,Z 597.763,A -85,B 0,C 180,E1 16069.08,E2 16069.08} C_VEL
LIN {X 0,Y 370.108,Z 573.956,A -85,B 0,C 180,E1 16067.998,E2 16067.998} C_VEL
LIN {X 0,Y 380.25,Z 515.563,A -85,B 0,C 180,E1 16065.905,E2 16065.905} C_VEL
LIN {X 0,Y 391.481,Z 464.537,A -85,B 0,C 180,E1 16064.069,E2 16064.069} C_VEL
LIN {X 0,Y 399.695,Z 432.421,A -85,B 0,C 180,E1 16062.925,E2 16062.925} C_VEL
LIN {X 0,Y 383.918,Z 497.009,A -85,B 0,C 180,E1 16060.574,E2 16060.574} C_VEL
LIN {X 0,Y 372.15,Z 555.463,A -85,B 0,C 180,E1 16058.349,E2 16058.349} C_VEL
LIN {X 0,Y 367.645,Z 579.27,A -85,B 0,C 180,E1 16057.335,E2 16057.335} C_VEL
LIN {X 0,Y 363.116,Z 600.549,A -85,B 0,C 180,E1 16056.104,E2 16056.104} C_VEL
LIN {X 0,Y 358.234,Z 621.939,A -85,B 0,C 180,E1 16054.512,E2 16054.512} C_VEL
LIN {X 0,Y 353.563,Z 641.476,A -85,B 0,C 180,E1 16052.692,E2 16052.692} C_VEL
LIN {X 0,Y 349.098,Z 659.317,A -85,B 0,C 180,E1 16050.651,E2 16050.651} C_VEL
LIN {X 0,Y 344.901,Z 675.585,A -85,B 0,C 180,E1 16048.387,E2 16048.387} C_VEL
LIN {X 0,Y 341.034,Z 690.337,A -85,B 0,C 180,E1 16045.902,E2 16045.902} C_VEL
LIN {X 0,Y 337.575,Z 703.545,A -85,B 0,C 180,E1 16043.199,E2 16043.199} C_VEL
LIN {X 0,Y 334.599,Z 715.171,A -85,B 0,C 180,E1 16040.281,E2 16040.281} C_VEL
LIN {X 0,Y 332.292,Z 724.649,A -85,B 0,C 180,E1 16037.33,E2 16037.33} C_VEL
LIN {X 0,Y 330.597,Z 732.231,A -85,B 0,C 180,E1 16034.359,E2 16034.359} C_VEL
LIN {X 0,Y 329.386,Z 738.403,A -85,B 0,C 180,E1 16031.202,E2 16031.202} C_VEL
LIN {X 0,Y 328.658,Z 742.803,A -85,B 0,C 180,E1 16028.044,E2 16028.044} C_VEL
LIN {X 0,Y 328.278,Z 745.629,A -85,B 0,C 180,E1 16024.716,E2 16024.716} C_VEL
LIN {X 0,Y 328.142,Z 746.633,A -85,B 0,C 180,E1 16021.571,E2 16021.571} C_VEL
LIN {X 0,Y 328.103,Z 746.012,A -85,B 0,C 180,E1 16018.428,E2 16018.428} C_VEL
LIN {X 0,Y 328.151,Z 743.758,A -85,B 0,C 180,E1 16015.28,E2 16015.28} C_VEL
LIN {X 0,Y 328.372,Z 739.807,A -85,B 0,C 180,E1 16012.124,E2 16012.124} C_VEL
LIN {X 0,Y 328.849,Z 734.444,A -85,B 0,C 180,E1 16009.133,E2 16009.133} C_VEL
LIN {X 0,Y 329.72,Z 727.043,A -85,B 0,C 180,E1 16006.025,E2 16006.025} C_VEL
LIN {X 0,Y 330.982,Z 718.343,A -85,B 0,C 180,E1 16003.141,E2 16003.141} C_VEL
LIN {X 0,Y 332.702,Z 707.869,A -85,B 0,C 180,E1 16000.33,E2 16000.33} C_VEL
LIN {X 0,Y 334.795,Z 695.999,A -85,B 0,C 180,E1 15997.71,E2 15997.71} C_VEL
LIN {X 0,Y 337.291,Z 682.225,A -85,B 0,C 180,E1 15995.199,E2 15995.199} C_VEL
LIN {X 0,Y 339.946,Z 667.484,A -85,B 0,C 180,E1 15992.972,E2 15992.972} C_VEL
LIN {X 0,Y 342.754,Z 651.22,A -85,B 0,C 180,E1 15990.941,E2 15990.941} C_VEL
LIN {X 0,Y 345.512,Z 634.102,A -85,B 0,C 180,E1 15989.188,E2 15989.188} C_VEL
LIN {X 0,Y 348.253,Z 615.141,A -85,B 0,C 180,E1 15987.624,E2 15987.624} C_VEL
LIN {X 0,Y 350.723,Z 595.391,A -85,B 0,C 180,E1 15986.353,E2 15986.353} C_VEL
LIN {X 0,Y 352.768,Z 575.246,A -85,B 0,C 180,E1 15985.382,E2 15985.382} C_VEL
LIN {X 0,Y 354.34,Z 554.645,A -85,B 0,C 180,E1 15984.694,E2 15984.694} C_VEL
LIN {X 0,Y 364.432,Z 383.187,A -85,B 0,C 180,E1 15980.267,E2 15980.267} C_VEL
LIN {X 0,Y 362.119,Z 366.133,A -85,B 0,C 180,E1 15979.436,E2 15979.436} C_VEL
LIN {X 0,Y 348.934,Z 341.464,A -85,B 0,C 180,E1 15976.946,E2 15976.946} C_VEL
LIN {X 0,Y 347.117,Z 337.74,A -85,B 0,C 180,E1 15976.493,E2 15976.493} C_VEL
LIN {X 0,Y 339.998,Z 319.459,A -85,B 0,C 180,E1 15972.792,E2 15972.792} C_VEL
LIN {X 0,Y 333.092,Z 302.809,A -85,B 0,C 180,E1 15969.079,E2 15969.079} C_VEL
LIN {X 0,Y 330.076,Z 295.57,A -85,B 0,C 180,E1 15967.285,E2 15967.285} C_VEL
LIN {X 0,Y 330.043,Z 295.371,A -85,B 0,C 180,E1 15962.946,E2 15962.946} C_VEL
LIN {X 0,Y 330.044,Z 295.349,A -85,B 0,C 180,E1 15958.531,E2 15958.531} C_VEL
LIN {X 0,Y 330.072,Z 295.561,A -85,B 0,C 180,E1 15956.347,E2 15956.347} C_VEL
LIN {X 0,Y 330.669,Z 297.596,A -85,B 0,C 180,E1 15955.897,E2 15955.897} C_VEL
LIN {X 0,Y 332.502,Z 301.305,A -85,B 0,C 180,E1 15955.157,E2 15955.157} C_VEL
LIN {X 0,Y 338.631,Z 314.413,A -85,B 0,C 180,E1 15952.665,E2 15952.665} C_VEL
LIN {X 0,Y 346.07,Z 332.865,A -85,B 0,C 180,E1 15949.504,E2 15949.504} C_VEL
LIN {X 0,Y 352.203,Z 350.651,A -85,B 0,C 180,E1 15946.749,E2 15946.749} C_VEL
LIN {X 0,Y 353.624,Z 356.013,A -85,B 0,C 180,E1 15945.982,E2 15945.982} C_VEL
LIN {X 0,Y 350.25,Z 397.698,A -85,B 0,C 180,E1 15941.812,E2 15941.812} C_VEL
LIN {X 0,Y 346.855,Z 438.589,A -85,B 0,C 180,E1 15937.705,E2 15937.705} C_VEL
LIN {X 0,Y 343.61,Z 481.813,A -85,B 0,C 180,E1 15933.411,E2 15933.411} C_VEL
LIN {X 0,Y 345.616,Z 502.462,A -85,B 0,C 180,E1 15932.753,E2 15932.753} C_VEL
LIN {X 0,Y 344.007,Z 560.903,A -85,B 0,C 180,E1 15931.522,E2 15931.522} C_VEL
LIN {X 0,Y 342.904,Z 568.569,A -85,B 0,C 180,E1 15931.431,E2 15931.431} C_VEL
LIN {X 0,Y 336.695,Z 588.888,A -85,B 0,C 180,E1 15931.446,E2 15931.446} C_VEL
LIN {X 0,Y 335.813,Z 595.472,A -85,B 0,C 180,E1 15931.361,E2 15931.361} C_VEL
LIN {X 0,Y 334.887,Z 627.398,A -85,B 0,C 180,E1 15930.611,E2 15930.611} C_VEL
LIN {X 0,Y 333.893,Z 644.369,A -85,B 0,C 180,E1 15929.868,E2 15929.868} C_VEL
LIN {X 0,Y 332.58,Z 659.659,A -85,B 0,C 180,E1 15928.882,E2 15928.882} C_VEL
LIN {X 0,Y 330.794,Z 675.437,A -85,B 0,C 180,E1 15927.49,E2 15927.49} C_VEL
LIN {X 0,Y 328.935,Z 689.154,A -85,B 0,C 180,E1 15925.906,E2 15925.906} C_VEL
LIN {X 0,Y 326.922,Z 702.47,A -85,B 0,C 180,E1 15923.945,E2 15923.945} C_VEL
LIN {X 0,Y 325.117,Z 713.568,A -85,B 0,C 180,E1 15921.869,E2 15921.869} C_VEL
LIN {X 0,Y 323.428,Z 723.844,A -85,B 0,C 180,E1 15919.449,E2 15919.449} C_VEL
LIN {X 0,Y 322.094,Z 732.194,A -85,B 0,C 180,E1 15916.905,E2 15916.905} C_VEL
LIN {X 0,Y 321.1,Z 739.181,A -85,B 0,C 180,E1 15914.099,E2 15914.099} C_VEL
LIN {X 0,Y 320.51,Z 744.121,A -85,B 0,C 180,E1 15911.26,E2 15911.26} C_VEL
LIN {X 0,Y 320.237,Z 747.308,A -85,B 0,C 180,E1 15908.384,E2 15908.384} C_VEL
LIN {X 0,Y 320.153,Z 748.689,A -85,B 0,C 180,E1 15905.46,E2 15905.46} C_VEL
LIN {X 0,Y 320.208,Z 748.308,A -85,B 0,C 180,E1 15902.475,E2 15902.475} C_VEL
LIN {X 0,Y 320.437,Z 746.187,A -85,B 0,C 180,E1 15899.639,E2 15899.639} C_VEL
LIN {X 0,Y 320.956,Z 742.246,A -85,B 0,C 180,E1 15896.753,E2 15896.753} C_VEL
LIN {X 0,Y 321.823,Z 736.738,A -85,B 0,C 180,E1 15894.045,E2 15894.045} C_VEL
LIN {X 0,Y 323.216,Z 728.85,A -85,B 0,C 180,E1 15891.221,E2 15891.221} C_VEL
LIN {X 0,Y 324.847,Z 719.976,A -85,B 0,C 180,E1 15888.804,E2 15888.804} C_VEL
LIN {X 0,Y 326.856,Z 709.046,A -85,B 0,C 180,E1 15886.469,E2 15886.469} C_VEL
LIN {X 0,Y 328.852,Z 697.514,A -85,B 0,C 180,E1 15884.525,E2 15884.525} C_VEL
LIN {X 0,Y 331.034,Z 683.779,A -85,B 0,C 180,E1 15882.694,E2 15882.694} C_VEL
LIN {X 0,Y 332.952,Z 669.65,A -85,B 0,C 180,E1 15881.238,E2 15881.238} C_VEL
LIN {X 0,Y 334.649,Z 654.366,A -85,B 0,C 180,E1 15880.042,E2 15880.042} C_VEL
LIN {X 0,Y 335.907,Z 638.471,A -85,B 0,C 180,E1 15879.155,E2 15879.155} C_VEL
LIN {X 0,Y 336.731,Z 621.67,A -85,B 0,C 180,E1 15878.553,E2 15878.553} C_VEL
LIN {X 0,Y 340.273,Z 500.964,A -85,B 0,C 180,E1 15875.903,E2 15875.903} C_VEL
LIN {X 0,Y 338.291,Z 482.445,A -85,B 0,C 180,E1 15875.195,E2 15875.195} C_VEL
LIN {X 0,Y 342.014,Z 438.182,A -85,B 0,C 180,E1 15870.745,E2 15870.745} C_VEL
LIN {X 0,Y 345.643,Z 397.177,A -85,B 0,C 180,E1 15866.643,E2 15866.643} C_VEL
LIN {X 0,Y 348.845,Z 358.991,A -85,B 0,C 180,E1 15862.854,E2 15862.854} C_VEL
LIN {X 0,Y 344.084,Z 343.766,A -85,B 0,C 180,E1 15860.409,E2 15860.409} C_VEL
LIN {X 0,Y 338.376,Z 328.993,A -85,B 0,C 180,E1 15857.72,E2 15857.72} C_VEL
LIN {X 0,Y 331.614,Z 314.432,A -85,B 0,C 180,E1 15854.672,E2 15854.672} C_VEL
LIN {X 0,Y 326.919,Z 305.633,A -85,B 0,C 180,E1 15852.542,E2 15852.542} C_VEL
LIN {X 0,Y 324.243,Z 300.882,A -85,B 0,C 180,E1 15851.316,E2 15851.316} C_VEL
LIN {X 0,Y 322.535,Z 298.193,A -85,B 0,C 180,E1 15850.539,E2 15850.539} C_VEL
LIN {X 0,Y 322.105,Z 296.499,A -85,B 0,C 180,E1 15850.011,E2 15850.011} C_VEL
LIN {X 0,Y 322.099,Z 296.361,A -85,B 0,C 180,E1 15845.702,E2 15845.702} C_VEL
LIN {X 0,Y 322.113,Z 296.356,A -85,B 0,C 180,E1 15841.246,E2 15841.246} C_VEL
LIN {X 0,Y 322.102,Z 296.36,A -85,B 0,C 180,E1 15836.976,E2 15836.976} C_VEL
LIN {X 0,Y 322.1,Z 296.357,A -85,B 0,C 180,E1 15832.689,E2 15832.689} C_VEL
LIN {X 0,Y 322.087,Z 296.364,A -85,B 0,C 180,E1 15828.36,E2 15828.36} C_VEL
LIN {X 0,Y 322.086,Z 296.356,A -85,B 0,C 180,E1 15823.962,E2 15823.962} C_VEL
LIN {X 0,Y 322.097,Z 296.365,A -85,B 0,C 180,E1 15819.624,E2 15819.624} C_VEL
LIN {X 0,Y 322.103,Z 296.358,A -85,B 0,C 180,E1 15815.421,E2 15815.421} C_VEL
LIN {X 0,Y 322.126,Z 296.358,A -85,B 0,C 180,E1 15811.04,E2 15811.04} C_VEL
LIN {X 0,Y 322.141,Z 296.599,A -85,B 0,C 180,E1 15807.255,E2 15807.255} C_VEL
LIN {X 0,Y 323.437,Z 299.898,A -85,B 0,C 180,E1 15806.403,E2 15806.403} C_VEL
LIN {X 0,Y 329.487,Z 313.282,A -85,B 0,C 180,E1 15803.287,E2 15803.287} C_VEL
LIN {X 0,Y 333.208,Z 321.551,A -85,B 0,C 180,E1 15801.549,E2 15801.549} C_VEL
LIN {X 0,Y 347.955,Z 346.12,A -85,B 0,C 180,E1 15798.521,E2 15798.521} C_VEL
LIN {X 0,Y 363.468,Z 373.851,A -85,B 0,C 180,E1 15795.604,E2 15795.604} C_VEL
LIN {X 0,Y 351.024,Z 576.718,A -85,B 0,C 180,E1 15790.451,E2 15790.451} C_VEL
LIN {X 0,Y 349.008,Z 597.716,A -85,B 0,C 180,E1 15789.646,E2 15789.646} C_VEL
LIN {X 0,Y 346.442,Z 618.576,A -85,B 0,C 180,E1 15788.545,E2 15788.545} C_VEL
LIN {X 0,Y 343.484,Z 638.791,A -85,B 0,C 180,E1 15787.155,E2 15787.155} C_VEL
LIN {X 0,Y 340.27,Z 658.146,A -85,B 0,C 180,E1 15785.482,E2 15785.482} C_VEL
LIN {X 0,Y 336.815,Z 677.039,A -85,B 0,C 180,E1 15783.471,E2 15783.471} C_VEL
LIN {X 0,Y 333.395,Z 694.677,A -85,B 0,C 180,E1 15781.178,E2 15781.178} C_VEL
LIN {X 0,Y 330.106,Z 711.106,A -85,B 0,C 180,E1 15778.589,E2 15778.589} C_VEL
LIN {X 0,Y 327.119,Z 726.145,A -85,B 0,C 180,E1 15775.721,E2 15775.721} C_VEL
LIN {X 0,Y 324.605,Z 739.455,A -85,B 0,C 180,E1 15772.643,E2 15772.643} C_VEL
LIN {X 0,Y 322.639,Z 751.062,A -85,B 0,C 180,E1 15769.363,E2 15769.363} C_VEL
LIN {X 0,Y 321.313,Z 760.445,A -85,B 0,C 180,E1 15766.076,E2 15766.076} C_VEL
LIN {X 0,Y 320.522,Z 767.872,A -85,B 0,C 180,E1 15762.794,E2 15762.794} C_VEL
LIN {X 0,Y 320.163,Z 773.545,A -85,B 0,C 180,E1 15759.525,E2 15759.525} C_VEL
LIN {X 0,Y 320.084,Z 777.59,A -85,B 0,C 180,E1 15756.275,E2 15756.275} C_VEL
LIN {X 0,Y 320.103,Z 780.047,A -85,B 0,C 180,E1 15753.042,E2 15753.042} C_VEL
LIN {X 0,Y 320.131,Z 780.898,A -85,B 0,C 180,E1 15749.819,E2 15749.819} C_VEL
LIN {X 0,Y 320.076,Z 780.269,A -85,B 0,C 180,E1 15746.595,E2 15746.595} C_VEL
LIN {X 0,Y 320.049,Z 778.155,A -85,B 0,C 180,E1 15743.36,E2 15743.36} C_VEL
LIN {X 0,Y 320.158,Z 774.434,A -85,B 0,C 180,E1 15740.108,E2 15740.108} C_VEL
LIN {X 0,Y 320.623,Z 768.833,A -85,B 0,C 180,E1 15736.646,E2 15736.646} C_VEL
LIN {X 0,Y 321.634,Z 761.444,A -85,B 0,C 180,E1 15733.194,E2 15733.194} C_VEL
LIN {X 0,Y 323.208,Z 752.634,A -85,B 0,C 180,E1 15729.915,E2 15729.915} C_VEL
LIN {X 0,Y 325.492,Z 741.846,A -85,B 0,C 180,E1 15726.653,E2 15726.653} C_VEL
LIN {X 0,Y 328.572,Z 728.823,A -85,B 0,C 180,E1 15723.426,E2 15723.426} C_VEL
LIN {X 0,Y 332.275,Z 714.126,A -85,B 0,C 180,E1 15720.416,E2 15720.416} C_VEL
LIN {X 0,Y 336.498,Z 697.928,A -85,B 0,C 180,E1 15717.665,E2 15717.665} C_VEL
LIN {X 0,Y 341.157,Z 680.064,A -85,B 0,C 180,E1 15715.143,E2 15715.143} C_VEL
LIN {X 0,Y 346.019,Z 661.29,A -85,B 0,C 180,E1 15712.95,E2 15712.95} C_VEL
LIN {X 0,Y 351.14,Z 641.007,A -85,B 0,C 180,E1 15711.001,E2 15711.001} C_VEL
LIN {X 0,Y 356.482,Z 619.129,A -85,B 0,C 180,E1 15709.297,E2 15709.297} C_VEL
LIN {X 0,Y 361.756,Z 596.519,A -85,B 0,C 180,E1 15707.912,E2 15707.912} C_VEL
LIN {X 0,Y 366.888,Z 572.676,A -85,B 0,C 180,E1 15706.812,E2 15706.812} C_VEL
LIN {X 0,Y 377.868,Z 517.801,A -85,B 0,C 180,E1 15704.793,E2 15704.793} C_VEL
LIN {X 0,Y 390.643,Z 466.175,A -85,B 0,C 180,E1 15702.92,E2 15702.92} C_VEL
LIN {X 0,Y 375.431,Z 527.422,A -85,B 0,C 180,E1 15700.616,E2 15700.616} C_VEL
LIN {X 0,Y 365.285,Z 574.697,A -85,B 0,C 180,E1 15698.715,E2 15698.715} C_VEL
LIN {X 0,Y 360.226,Z 596.098,A -85,B 0,C 180,E1 15697.535,E2 15697.535} C_VEL
LIN {X 0,Y 355.032,Z 616.708,A -85,B 0,C 180,E1 15696.057,E2 15696.057} C_VEL
LIN {X 0,Y 349.752,Z 636.453,A -85,B 0,C 180,E1 15694.275,E2 15694.275} C_VEL
LIN {X 0,Y 344.549,Z 655.366,A -85,B 0,C 180,E1 15692.174,E2 15692.174} C_VEL
LIN {X 0,Y 339.7,Z 672.619,A -85,B 0,C 180,E1 15689.829,E2 15689.829} C_VEL
LIN {X 0,Y 335.344,Z 687.875,A -85,B 0,C 180,E1 15687.31,E2 15687.31} C_VEL
LIN {X 0,Y 331.458,Z 701.373,A -85,B 0,C 180,E1 15684.6,E2 15684.6} C_VEL
LIN {X 0,Y 328.046,Z 713.374,A -85,B 0,C 180,E1 15681.641,E2 15681.641} C_VEL
LIN {X 0,Y 325.36,Z 723.236,A -85,B 0,C 180,E1 15678.638,E2 15678.638} C_VEL
LIN {X 0,Y 323.337,Z 731.206,A -85,B 0,C 180,E1 15675.606,E2 15675.606} C_VEL
LIN {X 0,Y 321.844,Z 737.757,A -85,B 0,C 180,E1 15672.377,E2 15672.377} C_VEL
LIN {X 0,Y 320.915,Z 742.528,A -85,B 0,C 180,E1 15669.142,E2 15669.142} C_VEL
LIN {X 0,Y 320.397,Z 745.718,A -85,B 0,C 180,E1 15665.731,E2 15665.731} C_VEL
LIN {X 0,Y 320.185,Z 747.083,A -85,B 0,C 180,E1 15662.505,E2 15662.505} C_VEL
LIN {X 0,Y 320.124,Z 746.801,A -85,B 0,C 180,E1 15659.284,E2 15659.284} C_VEL
LIN {X 0,Y 320.137,Z 744.879,A -85,B 0,C 180,E1 15656.059,E2 15656.059} C_VEL
LIN {X 0,Y 320.308,Z 741.283,A -85,B 0,C 180,E1 15652.827,E2 15652.827} C_VEL
LIN {X 0,Y 320.76,Z 735.921,A -85,B 0,C 180,E1 15649.583,E2 15649.583} C_VEL
LIN {X 0,Y 321.553,Z 729.098,A -85,B 0,C 180,E1 15646.513,E2 15646.513} C_VEL
LIN {X 0,Y 322.818,Z 720.405,A -85,B 0,C 180,E1 15643.443,E2 15643.443} C_VEL
LIN {X 0,Y 324.538,Z 710.111,A -85,B 0,C 180,E1 15640.521,E2 15640.521} C_VEL
LIN {X 0,Y 326.746,Z 697.947,A -85,B 0,C 180,E1 15637.7,E2 15637.7} C_VEL
LIN {X 0,Y 329.37,Z 683.992,A -85,B 0,C 180,E1 15635.041,E2 15635.041} C_VEL
LIN {X 0,Y 332.191,Z 668.881,A -85,B 0,C 180,E1 15632.676,E2 15632.676} C_VEL
LIN {X 0,Y 335.198,Z 652.054,A -85,B 0,C 180,E1 15630.515,E2 15630.515} C_VEL
LIN {X 0,Y 337.999,Z 635.314,A -85,B 0,C 180,E1 15628.752,E2 15628.752} C_VEL
LIN {X 0,Y 340.71,Z 617.38,A -85,B 0,C 180,E1 15627.217,E2 15627.217} C_VEL
LIN {X 0,Y 343.225,Z 598.27,A -85,B 0,C 180,E1 15625.925,E2 15625.925} C_VEL
LIN {X 0,Y 345.44,Z 577.827,A -85,B 0,C 180,E1 15624.88,E2 15624.88} C_VEL
LIN {X 0,Y 347.173,Z 556.743,A -85,B 0,C 180,E1 15624.129,E2 15624.129} C_VEL
LIN {X 0,Y 357.874,Z 384.361,A -85,B 0,C 180,E1 15619.551,E2 15619.551} C_VEL
LIN {X 0,Y 355.884,Z 369.657,A -85,B 0,C 180,E1 15618.818,E2 15618.818} C_VEL
LIN {X 0,Y 341.429,Z 342.54,A -85,B 0,C 180,E1 15615.999,E2 15615.999} C_VEL
LIN {X 0,Y 338.884,Z 337.675,A -85,B 0,C 180,E1 15615.395,E2 15615.395} C_VEL
LIN {X 0,Y 331.893,Z 319.885,A -85,B 0,C 180,E1 15611.657,E2 15611.657} C_VEL
LIN {X 0,Y 325.215,Z 303.882,A -85,B 0,C 180,E1 15607.946,E2 15607.946} C_VEL
LIN {X 0,Y 322.135,Z 296.54,A -85,B 0,C 180,E1 15606.069,E2 15606.069} C_VEL
LIN {X 0,Y 322.115,Z 296.361,A -85,B 0,C 180,E1 15601.642,E2 15601.642} C_VEL
LIN {X 0,Y 322.138,Z 296.597,A -85,B 0,C 180,E1 15597.548,E2 15597.548} C_VEL
LIN {X 0,Y 323.046,Z 299.275,A -85,B 0,C 180,E1 15596.95,E2 15596.95} C_VEL
LIN {X 0,Y 324.547,Z 302.103,A -85,B 0,C 180,E1 15596.338,E2 15596.338} C_VEL
LIN {X 0,Y 331.128,Z 316.025,A -85,B 0,C 180,E1 15593.587,E2 15593.587} C_VEL
LIN {X 0,Y 338.332,Z 333.564,A -85,B 0,C 180,E1 15590.474,E2 15590.474} C_VEL
LIN {X 0,Y 344.673,Z 351.685,A -85,B 0,C 180,E1 15587.561,E2 15587.561} C_VEL
LIN {X 0,Y 346.739,Z 358.83,A -85,B 0,C 180,E1 15586.503,E2 15586.503} C_VEL
LIN {X 0,Y 343.159,Z 400.438,A -85,B 0,C 180,E1 15582.282,E2 15582.282} C_VEL
LIN {X 0,Y 339.592,Z 442.338,A -85,B 0,C 180,E1 15578.041,E2 15578.041} C_VEL
LIN {X 0,Y 336.435,Z 482.085,A -85,B 0,C 180,E1 15574.039,E2 15574.039} C_VEL
LIN {X 0,Y 338.461,Z 503.375,A -85,B 0,C 180,E1 15573.344,E2 15573.344} C_VEL
LIN {X 0,Y 335.813,Z 595.472,A -85,B 0,C 180,E1 15571.361,E2 15571.361} C_VEL
LIN {X 0,Y 334.692,Z 603.149,A -85,B 0,C 180,E1 15571.277,E2 15571.277} C_VEL
LIN {X 0,Y 328.705,Z 622.369,A -85,B 0,C 180,E1 15571.273,E2 15571.273} C_VEL
LIN {X 0,Y 327.484,Z 629.952,A -85,B 0,C 180,E1 15571.095,E2 15571.095} C_VEL
LIN {X 0,Y 326.471,Z 645.96,A -85,B 0,C 180,E1 15570.353,E2 15570.353} C_VEL
LIN {X 0,Y 325.031,Z 661.476,A -85,B 0,C 180,E1 15569.297,E2 15569.297} C_VEL
